LIN {X 0,Y 333.342,Z 944.319,A -85,B 0,C 180,E1 -9784.98,E2 -9784.98} C_VEL
LIN {X 0,Y 331.25,Z 957.354,A -85,B 0,C 180,E1 -9788.578,E2 -9788.578} C_VEL
LIN {X 0,Y 329.876,Z 968.022,A -85,B 0,C 180,E1 -9792.173,E2 -9792.173} C_VEL
LIN {X 0,Y 329.125,Z 976.186,A -85,B 0,C 180,E1 -9795.575,E2 -9795.575} C_VEL
LIN {X 0,Y 328.812,Z 982.598,A -85,B 0,C 180,E1 -9798.955,E2 -9798.955} C_VEL
LIN {X 0,Y 328.744,Z 987.468,A -85,B 0,C 180,E1 -9802.485,E2 -9802.485} C_VEL
LIN {X 0,Y 328.81,Z 990.364,A -85,B 0,C 180,E1 -9805.64,E2 -9805.64} C_VEL
LIN {X 0,Y 328.851,Z 991.822,A -85,B 0,C 180,E1 -9808.954,E2 -9808.954} C_VEL
LIN {X 0,Y 328.808,Z 991.751,A -85,B 0,C 180,E1 -9812.265,E2 -9812.265} C_VEL
LIN {X 0,Y 328.709,Z 990.204,A -85,B 0,C 180,E1 -9815.41,E2 -9815.41} C_VEL
LIN {X 0,Y 328.63,Z 986.844,A -85,B 0,C 180,E1 -9818.926,E2 -9818.926} C_VEL
LIN {X 0,Y 328.762,Z 981.971,A -85,B 0,C 180,E1 -9822.291,E2 -9822.291} C_VEL
LIN {X 0,Y 329.291,Z 975.055,A -85,B 0,C 180,E1 -9825.859,E2 -9825.859} C_VEL
LIN {X 0,Y 330.353,Z 966.159,A -85,B 0,C 180,E1 -9829.446,E2 -9829.446} C_VEL
LIN {X 0,Y 332.113,Z 955.071,A -85,B 0,C 180,E1 -9833.04,E2 -9833.04} C_VEL
LIN {X 0,Y 334.527,Z 942.274,A -85,B 0,C 180,E1 -9836.445,E2 -9836.445} C_VEL
LIN {X 0,Y 337.738,Z 926.952,A -85,B 0,C 180,E1 -9839.825,E2 -9839.825} C_VEL
LIN {X 0,Y 341.327,Z 910.684,A -85,B 0,C 180,E1 -9842.814,E2 -9842.814} C_VEL
LIN {X 0,Y 345.387,Z 892.681,A -85,B 0,C 180,E1 -9845.582,E2 -9845.582} C_VEL
LIN {X 0,Y 349.323,Z 874.881,A -85,B 0,C 180,E1 -9847.876,E2 -9847.876} C_VEL
LIN {X 0,Y 353.782,Z 854.185,A -85,B 0,C 180,E1 -9850.118,E2 -9850.118} C_VEL
LIN {X 0,Y 357.815,Z 834.405,A -85,B 0,C 180,E1 -9851.901,E2 -9851.901} C_VEL
LIN {X 0,Y 361.825,Z 812.887,A -85,B 0,C 180,E1 -9853.478,E2 -9853.478} C_VEL
LIN {X 0,Y 365.405,Z 791.398,A -85,B 0,C 180,E1 -9854.741,E2 -9854.741} C_VEL
LIN {X 0,Y 368.714,Z 768.497,A -85,B 0,C 180,E1 -9855.786,E2 -9855.786} C_VEL
LIN {X 0,Y 371.277,Z 745.338,A -85,B 0,C 180,E1 -9856.575,E2 -9856.575} C_VEL
LIN {X 0,Y 373.467,Z 717.783,A -85,B 0,C 180,E1 -9857.235,E2 -9857.235} C_VEL
LIN {X 0,Y 375.217,Z 704.776,A -85,B 0,C 180,E1 -9857.459,E2 -9857.459} C_VEL
LIN {X 0,Y 386.824,Z 676.005,A -85,B 0,C 180,E1 -9858.891,E2 -9858.891} C_VEL
LIN {X 0,Y 396.456,Z 655.426,A -85,B 0,C 180,E1 -9859.72,E2 -9859.72} C_VEL
LIN {X 0,Y 403.864,Z 640.656,A -85,B 0,C 180,E1 -9860.238,E2 -9860.238} C_VEL
LIN {X 0,Y 409.262,Z 629.343,A -85,B 0,C 180,E1 -9860.656,E2 -9860.656} C_VEL
LIN {X 0,Y 402.007,Z 613.046,A -85,B 0,C 180,E1 -9863.084,E2 -9863.084} C_VEL
LIN {X 0,Y 396.941,Z 595.631,A -85,B 0,C 180,E1 -9865.476,E2 -9865.476} C_VEL
LIN {X 0,Y 393.973,Z 576.533,A -85,B 0,C 180,E1 -9867.881,E2 -9867.881} C_VEL
LIN {X 0,Y 393.144,Z 556.331,A -85,B 0,C 180,E1 -9870.185,E2 -9870.185} C_VEL
LIN {X 0,Y 394.303,Z 535.428,A -85,B 0,C 180,E1 -9872.352,E2 -9872.352} C_VEL
LIN {X 0,Y 397.843,Z 510.824,A -85,B 0,C 180,E1 -9874.628,E2 -9874.628} C_VEL
LIN {X 0,Y 397.962,Z 509.912,A -85,B 0,C 180,E1 -9874.716,E2 -9874.716} C_VEL
LIN {X 0,Y 388.741,Z 492.166,A -85,B 0,C 180,E1 -9878.579,E2 -9878.579} C_VEL
LIN {X 0,Y 379.957,Z 475.806,A -85,B 0,C 180,E1 -9882.543,E2 -9882.543} C_VEL
LIN {X 0,Y 371.539,Z 460.665,A -85,B 0,C 180,E1 -9886.619,E2 -9886.619} C_VEL
LIN {X 0,Y 363.758,Z 446.974,A -85,B 0,C 180,E1 -9890.667,E2 -9890.667} C_VEL
LIN {X 0,Y 357.078,Z 435.672,A -85,B 0,C 180,E1 -9894.376,E2 -9894.376} C_VEL
LIN {X 0,Y 353.868,Z 430.258,A -85,B 0,C 180,E1 -9896.274,E2 -9896.274} C_VEL
LIN {X 0,Y 350.952,Z 425.333,A -85,B 0,C 180,E1 -9898.041,E2 -9898.041} C_VEL
LIN {X 0,Y 348.106,Z 420.507,A -85,B 0,C 180,E1 -9899.836,E2 -9899.836} C_VEL
LIN {X 0,Y 345.35,Z 415.775,A -85,B 0,C 180,E1 -9901.66,E2 -9901.66} C_VEL
LIN {X 0,Y 342.391,Z 410.76,A -85,B 0,C 180,E1 -9903.684,E2 -9903.684} C_VEL
LIN {X 0,Y 340.137,Z 407.168,A -85,B 0,C 180,E1 -9905.229,E2 -9905.229} C_VEL
LIN {X 0,Y 339.237,Z 405.463,A -85,B 0,C 180,E1 -9905.922,E2 -9905.922} C_VEL
LIN {X 0,Y 336.904,Z 401.699,A -85,B 0,C 180,E1 -9907.592,E2 -9907.592} C_VEL
LIN {X 0,Y 336.153,Z 400.24,A -85,B 0,C 180,E1 -9908.209,E2 -9908.209} C_VEL
LIN {X 0,Y 333.851,Z 396.936,A -85,B 0,C 180,E1 -9909.83,E2 -9909.83} C_VEL
LIN {X 0,Y 333.176,Z 395.055,A -85,B 0,C 180,E1 -9910.549,E2 -9910.549} C_VEL
LIN {X 0,Y 330.607,Z 391.768,A -85,B 0,C 180,E1 -9912.354,E2 -9912.354} C_VEL
LIN {X 0,Y 330.054,Z 389.618,A -85,B 0,C 180,E1 -9913.133,E2 -9913.133} C_VEL
LIN {X 0,Y 330.032,Z 389.621,A -85,B 0,C 180,E1 -9917.454,E2 -9917.454} C_VEL
LIN {X 0,Y 330.06,Z 389.619,A -85,B 0,C 180,E1 -9921.877,E2 -9921.877} C_VEL
LIN {X 0,Y 330.024,Z 389.616,A -85,B 0,C 180,E1 -9926.263,E2 -9926.263} C_VEL
LIN {X 0,Y 330.052,Z 389.609,A -85,B 0,C 180,E1 -9930.594,E2 -9930.594} C_VEL
LIN {X 0,Y 330.06,Z 389.802,A -85,B 0,C 180,E1 -9932.363,E2 -9932.363} C_VEL
LIN {X 0,Y 331.04,Z 392.665,A -85,B 0,C 180,E1 -9932.934,E2 -9932.934} C_VEL
LIN {X 0,Y 333.496,Z 395.723,A -85,B 0,C 180,E1 -9933.894,E2 -9933.894} C_VEL
LIN {X 0,Y 335.781,Z 399.63,A -85,B 0,C 180,E1 -9934.871,E2 -9934.871} C_VEL
LIN {X 0,Y 336.928,Z 401.545,A -85,B 0,C 180,E1 -9935.358,E2 -9935.358} C_VEL
LIN {X 0,Y 340.103,Z 406.895,A -85,B 0,C 180,E1 -9936.641,E2 -9936.641} C_VEL
LIN {X 0,Y 346.837,Z 418.945,A -85,B 0,C 180,E1 -9939.362,E2 -9939.362} C_VEL
LIN {X 0,Y 354.009,Z 433.623,A -85,B 0,C 180,E1 -9942.27,E2 -9942.27} C_VEL
LIN {X 0,Y 361.242,Z 450.647,A -85,B 0,C 180,E1 -9945.232,E2 -9945.232} C_VEL
LIN {X 0,Y 366.814,Z 465.9,A -85,B 0,C 180,E1 -9947.592,E2 -9947.592} C_VEL
LIN {X 0,Y 364.449,Z 505.857,A -85,B 0,C 180,E1 -9950.778,E2 -9950.778} C_VEL
LIN {X 0,Y 365.241,Z 514.351,A -85,B 0,C 180,E1 -9951.097,E2 -9951.097} C_VEL
LIN {X 0,Y 358.254,Z 708.662,A -85,B 0,C 180,E1 -9955.043,E2 -9955.043} C_VEL
LIN {X 0,Y 357.559,Z 727.861,A -85,B 0,C 180,E1 -9955.656,E2 -9955.656} C_VEL
LIN {X 0,Y 356.255,Z 746.186,A -85,B 0,C 180,E1 -9956.531,E2 -9956.531} C_VEL
LIN {X 0,Y 354.36,Z 763.972,A -85,B 0,C 180,E1 -9957.677,E2 -9957.677} C_VEL
LIN {X 0,Y 352.024,Z 780.749,A -85,B 0,C 180,E1 -9959.069,E2 -9959.069} C_VEL
LIN {X 0,Y 349.422,Z 796.485,A -85,B 0,C 180,E1 -9960.705,E2 -9960.705} C_VEL
LIN {X 0,Y 346.547,Z 811.319,A -85,B 0,C 180,E1 -9962.601,E2 -9962.601} C_VEL
LIN {X 0,Y 343.447,Z 825.625,A -85,B 0,C 180,E1 -9964.847,E2 -9964.847} C_VEL
LIN {X 0,Y 340.599,Z 837.864,A -85,B 0,C 180,E1 -9967.202,E2 -9967.202} C_VEL
LIN {X 0,Y 337.942,Z 848.709,A -85,B 0,C 180,E1 -9969.748,E2 -9969.748} C_VEL
LIN {X 0,Y 335.601,Z 858.18,A -85,B 0,C 180,E1 -9972.488,E2 -9972.488} C_VEL
LIN {X 0,Y 333.603,Z 866.416,A -85,B 0,C 180,E1 -9975.486,E2 -9975.486} C_VEL
LIN {X 0,Y 332.093,Z 872.879,A -85,B 0,C 180,E1 -9978.539,E2 -9978.539} C_VEL
LIN {X 0,Y 331.064,Z 877.731,A -85,B 0,C 180,E1 -9981.665,E2 -9981.665} C_VEL
LIN {X 0,Y 330.433,Z 881.111,A -85,B 0,C 180,E1 -9984.966,E2 -9984.966} C_VEL
LIN {X 0,Y 330.13,Z 882.813,A -85,B 0,C 180,E1 -9988.265,E2 -9988.265} C_VEL
LIN {X 0,Y 330.118,Z 882.889,A -85,B 0,C 180,E1 -9991.563,E2 -9991.563} C_VEL
LIN {X 0,Y 330.401,Z 881.34,A -85,B 0,C 180,E1 -9994.861,E2 -9994.861} C_VEL
LIN {X 0,Y 331.005,Z 878.106,A -85,B 0,C 180,E1 -9998.162,E2 -9998.162} C_VEL
LIN {X 0,Y 332.063,Z 873.069,A -85,B 0,C 180,E1 -10001.463,E2 -10001.463} C_VEL
LIN {X 0,Y 332.526,Z 871.056,A -85,B 0,C 180,E1 -10002.525,E2 -10002.525} C_VEL
LIN {X 0,Y 332.193,Z 868.673,A -85,B 0,C 180,E1 -10003.798,E2 -10003.798} C_VEL
LIN {X 0,Y 328.296,Z 862.096,A -85,B 0,C 180,E1 -10007.032,E2 -10007.032} C_VEL
LIN {X 0,Y 328.253,Z 858.758,A -85,B 0,C 180,E1 -10008.258,E2 -10008.258} C_VEL
LIN {X 0,Y 330.797,Z 849.028,A -85,B 0,C 180,E1 -10011.081,E2 -10011.081} C_VEL
LIN {X 0,Y 333.638,Z 837.979,A -85,B 0,C 180,E1 -10013.677,E2 -10013.677} C_VEL
LIN {X 0,Y 336.672,Z 825.502,A -85,B 0,C 180,E1 -10016.075,E2 -10016.075} C_VEL
LIN {X 0,Y 339.828,Z 811.487,A -85,B 0,C 180,E1 -10018.275,E2 -10018.275} C_VEL
LIN {X 0,Y 342.858,Z 796.414,A -85,B 0,C 180,E1 -10020.203,E2 -10020.203} C_VEL
LIN {X 0,Y 345.598,Z 780.325,A -85,B 0,C 180,E1 -10021.871,E2 -10021.871} C_VEL
LIN {X 0,Y 348.05,Z 763.099,A -85,B 0,C 180,E1 -10023.282,E2 -10023.282} C_VEL
LIN {X 0,Y 349.961,Z 744.96,A -85,B 0,C 180,E1 -10024.424,E2 -10024.424} C_VEL
LIN {X 0,Y 351.23,Z 726.587,A -85,B 0,C 180,E1 -10025.271,E2 -10025.271} C_VEL
LIN {X 0,Y 351.888,Z 707.076,A -85,B 0,C 180,E1 -10025.865,E2 -10025.865} C_VEL
LIN {X 0,Y 359.08,Z 513.009,A -85,B 0,C 180,E1 -10029.877,E2 -10029.877} C_VEL
LIN {X 0,Y 358.387,Z 506.854,A -85,B 0,C 180,E1 -10030.143,E2 -10030.143} C_VEL
LIN {X 0,Y 360.731,Z 469.551,A -85,B 0,C 180,E1 -10033.141,E2 -10033.141} C_VEL
LIN {X 0,Y 359.899,Z 467.043,A -85,B 0,C 180,E1 -10033.522,E2 -10033.522} C_VEL
LIN {X 0,Y 357.571,Z 466.596,A -85,B 0,C 180,E1 -10033.99,E2 -10033.99} C_VEL
LIN {X 0,Y 361.006,Z 476.688,A -85,B 0,C 180,E1 -10035.836,E2 -10035.836} C_VEL
LIN {X 0,Y 354.597,Z 519.378,A -85,B 0,C 180,E1 -10040.307,E2 -10040.307} C_VEL
LIN {X 0,Y 348.6,Z 563.579,A -85,B 0,C 180,E1 -10044.884,E2 -10044.884} C_VEL
LIN {X 0,Y 343.147,Z 608.894,A -85,B 0,C 180,E1 -10049.535,E2 -10049.535} C_VEL
LIN {X 0,Y 342.926,Z 612.486,A -85,B 0,C 180,E1 -10049.847,E2 -10049.847} C_VEL
LIN {X 0,Y 343.393,Z 622.189,A -85,B 0,C 180,E1 -10050.252,E2 -10050.252} C_VEL
LIN {X 0,Y 335.087,Z 752.809,A -85,B 0,C 180,E1 -10054.515,E2 -10054.515} C_VEL
LIN {X 0,Y 334.283,Z 770.76,A -85,B 0,C 180,E1 -10055.291,E2 -10055.291} C_VEL
LIN {X 0,Y 333.102,Z 788.151,A -85,B 0,C 180,E1 -10056.376,E2 -10056.376} C_VEL
LIN {X 0,Y 331.637,Z 804.493,A -85,B 0,C 180,E1 -10057.757,E2 -10057.757} C_VEL
LIN {X 0,Y 330.089,Z 819.19,A -85,B 0,C 180,E1 -10059.336,E2 -10059.336} C_VEL
LIN {X 0,Y 328.346,Z 834.099,A -85,B 0,C 180,E1 -10061.352,E2 -10061.352} C_VEL
LIN {X 0,Y 326.786,Z 846.627,A -85,B 0,C 180,E1 -10063.468,E2 -10063.468} C_VEL
LIN {X 0,Y 325.423,Z 857.745,A -85,B 0,C 180,E1 -10065.77,E2 -10065.77} C_VEL
LIN {X 0,Y 324.292,Z 867.369,A -85,B 0,C 180,E1 -10068.258,E2 -10068.258} C_VEL
LIN {X 0,Y 323.451,Z 875.603,A -85,B 0,C 180,E1 -10070.929,E2 -10070.929} C_VEL
LIN {X 0,Y 322.92,Z 882.228,A -85,B 0,C 180,E1 -10073.778,E2 -10073.778} C_VEL
LIN {X 0,Y 322.755,Z 887.037,A -85,B 0,C 180,E1 -10076.625,E2 -10076.625} C_VEL
LIN {X 0,Y 322.919,Z 890.358,A -85,B 0,C 180,E1 -10079.822,E2 -10079.822} C_VEL
LIN {X 0,Y 323.359,Z 891.535,A -85,B 0,C 180,E1 -10082.658,E2 -10082.658} C_VEL
LIN {X 0,Y 324.226,Z 891.056,A -85,B 0,C 180,E1 -10085.663,E2 -10085.663} C_VEL
LIN {X 0,Y 325.623,Z 888.514,A -85,B 0,C 180,E1 -10088.831,E2 -10088.831} C_VEL
LIN {X 0,Y 327.391,Z 884.461,A -85,B 0,C 180,E1 -10091.628,E2 -10091.628} C_VEL
LIN {X 0,Y 329.667,Z 878.673,A -85,B 0,C 180,E1 -10094.4,E2 -10094.4} C_VEL
LIN {X 0,Y 332.687,Z 870.277,A -85,B 0,C 180,E1 -10097.309,E2 -10097.309} C_VEL
LIN {X 0,Y 335.956,Z 860.542,A -85,B 0,C 180,E1 -10099.868,E2 -10099.868} C_VEL
LIN {X 0,Y 339.403,Z 849.527,A -85,B 0,C 180,E1 -10102.152,E2 -10102.152} C_VEL
LIN {X 0,Y 343.232,Z 836.315,A -85,B 0,C 180,E1 -10104.343,E2 -10104.343} C_VEL
LIN {X 0,Y 347.06,Z 821.915,A -85,B 0,C 180,E1 -10106.245,E2 -10106.245} C_VEL
LIN {X 0,Y 351.022,Z 805.964,A -85,B 0,C 180,E1 -10107.941,E2 -10107.941} C_VEL
LIN {X 0,Y 357.078,Z 783.037,A -85,B 0,C 180,E1 -10109.895,E2 -10109.895} C_VEL
LIN {X 0,Y 365.991,Z 756.399,A -85,B 0,C 180,E1 -10111.82,E2 -10111.82} C_VEL
LIN {X 0,Y 377.505,Z 723.16,A -85,B 0,C 180,E1 -10113.73,E2 -10113.73} C_VEL
LIN {X 0,Y 386.645,Z 693.172,A -85,B 0,C 180,E1 -10115.16,E2 -10115.16} C_VEL
LIN {X 0,Y 394.084,Z 667.225,A -85,B 0,C 180,E1 -10116.239,E2 -10116.239} C_VEL
LIN {X 0,Y 401.871,Z 655.163,A -85,B 0,C 180,E1 -10116.931,E2 -10116.931} C_VEL
LIN {X 0,Y 408.346,Z 646.955,A -85,B 0,C 180,E1 -10118.125,E2 -10118.125} C_VEL
LIN {X 0,Y 393.564,Z 674.807,A -85,B 0,C 180,E1 -10119.092,E2 -10119.092} C_VEL
LIN {X 0,Y 390.576,Z 686.577,A -85,B 0,C 180,E1 -10119.459,E2 -10119.459} C_VEL
LIN {X 0,Y 384.525,Z 712.431,A -85,B 0,C 180,E1 -10120.042,E2 -10120.042} C_VEL
LIN {X 0,Y 379.962,Z 730.467,A -85,B 0,C 180,E1 -10120.534,E2 -10120.534} C_VEL
LIN {X 0,Y 372.781,Z 758.728,A -85,B 0,C 180,E1 -10121.785,E2 -10121.785} C_VEL
LIN {X 0,Y 365.463,Z 785.63,A -85,B 0,C 180,E1 -10123.302,E2 -10123.302} C_VEL
LIN {X 0,Y 358.515,Z 810.818,A -85,B 0,C 180,E1 -10125.122,E2 -10125.122} C_VEL
LIN {X 0,Y 351.985,Z 834.7,A -85,B 0,C 180,E1 -10127.241,E2 -10127.241} C_VEL
LIN {X 0,Y 345.36,Z 859.368,A -85,B 0,C 180,E1 -10129.896,E2 -10129.896} C_VEL
LIN {X 0,Y 340.054,Z 879.999,A -85,B 0,C 180,E1 -10132.549,E2 -10132.549} C_VEL
LIN {X 0,Y 335.233,Z 899.403,A -85,B 0,C 180,E1 -10135.48,E2 -10135.48} C_VEL
LIN {X 0,Y 331.225,Z 916.555,A -85,B 0,C 180,E1 -10138.517,E2 -10138.517} C_VEL
LIN {X 0,Y 327.784,Z 932.46,A -85,B 0,C 180,E1 -10141.829,E2 -10141.829} C_VEL
LIN {X 0,Y 324.959,Z 947.091,A -85,B 0,C 180,E1 -10145.456,E2 -10145.456} C_VEL
LIN {X 0,Y 322.917,Z 959.714,A -85,B 0,C 180,E1 -10149.242,E2 -10149.242} C_VEL
LIN {X 0,Y 321.657,Z 969.925,A -85,B 0,C 180,E1 -10153.01,E2 -10153.01} C_VEL
LIN {X 0,Y 321.02,Z 977.806,A -85,B 0,C 180,E1 -10156.674,E2 -10156.674} C_VEL
LIN {X 0,Y 320.802,Z 983.523,A -85,B 0,C 180,E1 -10160.129,E2 -10160.129} C_VEL
LIN {X 0,Y 320.84,Z 987.541,A -85,B 0,C 180,E1 -10163.558,E2 -10163.558} C_VEL
LIN {X 0,Y 320.909,Z 989.98,A -85,B 0,C 180,E1 -10166.963,E2 -10166.963} C_VEL
LIN {X 0,Y 320.944,Z 990.779,A -85,B 0,C 180,E1 -10170.178,E2 -10170.178} C_VEL
LIN {X 0,Y 320.86,Z 990.107,A -85,B 0,C 180,E1 -10173.573,E2 -10173.573} C_VEL
LIN {X 0,Y 320.719,Z 987.806,A -85,B 0,C 180,E1 -10176.983,E2 -10176.983} C_VEL
LIN {X 0,Y 320.715,Z 983.933,A -85,B 0,C 180,E1 -10180.417,E2 -10180.417} C_VEL
LIN {X 0,Y 320.994,Z 978.022,A -85,B 0,C 180,E1 -10184.061,E2 -10184.061} C_VEL
LIN {X 0,Y 321.719,Z 970.64,A -85,B 0,C 180,E1 -10187.545,E2 -10187.545} C_VEL
LIN {X 0,Y 323.027,Z 961.408,A -85,B 0,C 180,E1 -10191.042,E2 -10191.042} C_VEL
LIN {X 0,Y 325.146,Z 949.445,A -85,B 0,C 180,E1 -10194.721,E2 -10194.721} C_VEL
LIN {X 0,Y 327.969,Z 935.671,A -85,B 0,C 180,E1 -10198.199,E2 -10198.199} C_VEL
LIN {X 0,Y 331.295,Z 920.762,A -85,B 0,C 180,E1 -10201.34,E2 -10201.34} C_VEL
LIN {X 0,Y 335.216,Z 903.919,A -85,B 0,C 180,E1 -10204.314,E2 -10204.314} C_VEL
LIN {X 0,Y 339.551,Z 885.243,A -85,B 0,C 180,E1 -10207.061,E2 -10207.061} C_VEL
LIN {X 0,Y 344.261,Z 864.347,A -85,B 0,C 180,E1 -10209.601,E2 -10209.601} C_VEL
LIN {X 0,Y 348.606,Z 844.573,A -85,B 0,C 180,E1 -10211.604,E2 -10211.604} C_VEL
LIN {X 0,Y 352.957,Z 823.133,A -85,B 0,C 180,E1 -10213.389,E2 -10213.389} C_VEL
LIN {X 0,Y 356.828,Z 801.846,A -85,B 0,C 180,E1 -10214.819,E2 -10214.819} C_VEL
LIN {X 0,Y 360.627,Z 778.349,A -85,B 0,C 180,E1 -10216.057,E2 -10216.057} C_VEL
LIN {X 0,Y 363.715,Z 755.272,A -85,B 0,C 180,E1 -10216.972,E2 -10216.972} C_VEL
LIN {X 0,Y 365.801,Z 731.561,A -85,B 0,C 180,E1 -10217.667,E2 -10217.667} C_VEL
LIN {X 0,Y 367.996,Z 710.151,A -85,B 0,C 180,E1 -10218.106,E2 -10218.106} C_VEL
LIN {X 0,Y 368.838,Z 704.318,A -85,B 0,C 180,E1 -10218.2,E2 -10218.2} C_VEL
LIN {X 0,Y 380.549,Z 675.592,A -85,B 0,C 180,E1 -10219.636,E2 -10219.636} C_VEL
LIN {X 0,Y 390.175,Z 655.218,A -85,B 0,C 180,E1 -10220.474,E2 -10220.474} C_VEL
LIN {X 0,Y 398.096,Z 639.628,A -85,B 0,C 180,E1 -10221.017,E2 -10221.017} C_VEL
LIN {X 0,Y 401.859,Z 631.602,A -85,B 0,C 180,E1 -10221.325,E2 -10221.325} C_VEL
LIN {X 0,Y 394.83,Z 614.668,A -85,B 0,C 180,E1 -10223.84,E2 -10223.84} C_VEL
LIN {X 0,Y 390.221,Z 597.312,A -85,B 0,C 180,E1 -10226.22,E2 -10226.22} C_VEL
LIN {X 0,Y 387.565,Z 578.081,A -85,B 0,C 180,E1 -10228.641,E2 -10228.641} C_VEL
LIN {X 0,Y 387.071,Z 557.241,A -85,B 0,C 180,E1 -10231.031,E2 -10231.031} C_VEL
LIN {X 0,Y 388.574,Z 535.98,A -85,B 0,C 180,E1 -10233.237,E2 -10233.237} C_VEL
LIN {X 0,Y 391.857,Z 514.196,A -85,B 0,C 180,E1 -10235.263,E2 -10235.263} C_VEL
LIN {X 0,Y 383.368,Z 497.684,A -85,B 0,C 180,E1 -10238.905,E2 -10238.905} C_VEL
LIN {X 0,Y 374.539,Z 481.229,A -85,B 0,C 180,E1 -10242.924,E2 -10242.924} C_VEL
LIN {X 0,Y 366.427,Z 466.54,A -85,B 0,C 180,E1 -10246.911,E2 -10246.911} C_VEL
LIN {X 0,Y 358.659,Z 452.809,A -85,B 0,C 180,E1 -10251.019,E2 -10251.019} C_VEL
LIN {X 0,Y 351.921,Z 441.384,A -85,B 0,C 180,E1 -10254.784,E2 -10254.784} C_VEL
LIN {X 0,Y 348.681,Z 435.902,A -85,B 0,C 180,E1 -10256.713,E2 -10256.713} C_VEL
LIN {X 0,Y 345.807,Z 430.994,A -85,B 0,C 180,E1 -10258.509,E2 -10258.509} C_VEL
LIN {X 0,Y 343.227,Z 426.58,A -85,B 0,C 180,E1 -10260.167,E2 -10260.167} C_VEL
LIN {X 0,Y 340.412,Z 421.817,A -85,B 0,C 180,E1 -10262.02,E2 -10262.02} C_VEL
LIN {X 0,Y 337.395,Z 416.778,A -85,B 0,C 180,E1 -10264.079,E2 -10264.079} C_VEL
LIN {X 0,Y 335.066,Z 412.505,A -85,B 0,C 180,E1 -10265.824,E2 -10265.824} C_VEL
LIN {X 0,Y 332.326,Z 408.24,A -85,B 0,C 180,E1 -10267.782,E2 -10267.782} C_VEL
LIN {X 0,Y 331.376,Z 406.559,A -85,B 0,C 180,E1 -10268.503,E2 -10268.503} C_VEL
LIN {X 0,Y 328.991,Z 402.694,A -85,B 0,C 180,E1 -10270.33,E2 -10270.33} C_VEL
LIN {X 0,Y 328.052,Z 401.087,A -85,B 0,C 180,E1 -10271.067,E2 -10271.067} C_VEL
LIN {X 0,Y 325.86,Z 397.789,A -85,B 0,C 180,E1 -10272.764,E2 -10272.764} C_VEL
LIN {X 0,Y 325.032,Z 395.848,A -85,B 0,C 180,E1 -10273.574,E2 -10273.574} C_VEL
LIN {X 0,Y 322.788,Z 392.975,A -85,B 0,C 180,E1 -10275.266,E2 -10275.266} C_VEL
LIN {X 0,Y 322.094,Z 390.61,A -85,B 0,C 180,E1 -10276.224,E2 -10276.224} C_VEL
LIN {X 0,Y 322.11,Z 390.604,A -85,B 0,C 180,E1 -10280.915,E2 -10280.915} C_VEL
LIN {X 0,Y 322.083,Z 390.617,A -85,B 0,C 180,E1 -10285.397,E2 -10285.397} C_VEL
LIN {X 0,Y 322.114,Z 390.612,A -85,B 0,C 180,E1 -10289.643,E2 -10289.643} C_VEL
LIN {X 0,Y 322.126,Z 390.626,A -85,B 0,C 180,E1 -10290.312,E2 -10290.312} C_VEL
LIN {X 0,Y 323.043,Z 393.495,A -85,B 0,C 180,E1 -10290.917,E2 -10290.917} C_VEL
LIN {X 0,Y 325.472,Z 396.18,A -85,B 0,C 180,E1 -10291.897,E2 -10291.897} C_VEL
LIN {X 0,Y 327.525,Z 400.234,A -85,B 0,C 180,E1 -10292.916,E2 -10292.916} C_VEL
LIN {X 0,Y 329.128,Z 402.367,A -85,B 0,C 180,E1 -10293.567,E2 -10293.567} C_VEL
LIN {X 0,Y 332.527,Z 408.079,A -85,B 0,C 180,E1 -10295.052,E2 -10295.052} C_VEL
LIN {X 0,Y 337.194,Z 416.006,A -85,B 0,C 180,E1 -10297.01,E2 -10297.01} C_VEL
LIN {X 0,Y 344.143,Z 429.404,A -85,B 0,C 180,E1 -10299.948,E2 -10299.948} C_VEL
LIN {X 0,Y 350.801,Z 443.734,A -85,B 0,C 180,E1 -10302.716,E2 -10302.716} C_VEL
LIN {X 0,Y 357.748,Z 461.185,A -85,B 0,C 180,E1 -10305.684,E2 -10305.684} C_VEL
LIN {X 0,Y 360.649,Z 469.904,A -85,B 0,C 180,E1 -10307,E2 -10307} C_VEL
LIN {X 0,Y 358.347,Z 507.3,A -85,B 0,C 180,E1 -10309.985,E2 -10309.985} C_VEL
LIN {X 0,Y 359.086,Z 515.499,A -85,B 0,C 180,E1 -10310.3,E2 -10310.3} C_VEL
LIN {X 0,Y 351.79,Z 709.225,A -85,B 0,C 180,E1 -10314.288,E2 -10314.288} C_VEL
LIN {X 0,Y 351.081,Z 728.581,A -85,B 0,C 180,E1 -10314.906,E2 -10314.906} C_VEL
LIN {X 0,Y 349.757,Z 746.717,A -85,B 0,C 180,E1 -10315.775,E2 -10315.775} C_VEL
LIN {X 0,Y 347.856,Z 764.136,A -85,B 0,C 180,E1 -10316.899,E2 -10316.899} C_VEL
LIN {X 0,Y 345.564,Z 780.231,A -85,B 0,C 180,E1 -10318.224,E2 -10318.224} C_VEL
LIN {X 0,Y 342.826,Z 796.335,A -85,B 0,C 180,E1 -10319.892,E2 -10319.892} C_VEL
LIN {X 0,Y 339.769,Z 811.562,A -85,B 0,C 180,E1 -10321.84,E2 -10321.84} C_VEL
LIN {X 0,Y 336.765,Z 824.956,A -85,B 0,C 180,E1 -10323.934,E2 -10323.934} C_VEL
LIN {X 0,Y 333.72,Z 837.525,A -85,B 0,C 180,E1 -10326.33,E2 -10326.33} C_VEL
LIN {X 0,Y 330.869,Z 848.651,A -85,B 0,C 180,E1 -10328.924,E2 -10328.924} C_VEL
LIN {X 0,Y 328.332,Z 858.368,A -85,B 0,C 180,E1 -10331.72,E2 -10331.72} C_VEL
LIN {X 0,Y 326.085,Z 867.09,A -85,B 0,C 180,E1 -10334.893,E2 -10334.893} C_VEL
LIN {X 0,Y 324.408,Z 873.817,A -85,B 0,C 180,E1 -10338.083,E2 -10338.083} C_VEL
LIN {X 0,Y 323.28,Z 878.762,A -85,B 0,C 180,E1 -10341.284,E2 -10341.284} C_VEL
LIN {X 0,Y 322.582,Z 882.228,A -85,B 0,C 180,E1 -10344.665,E2 -10344.665} C_VEL
LIN {X 0,Y 322.242,Z 884.013,A -85,B 0,C 180,E1 -10348.045,E2 -10348.045} C_VEL
LIN {X 0,Y 322.209,Z 884.173,A -85,B 0,C 180,E1 -10351.423,E2 -10351.423} C_VEL
LIN {X 0,Y 322.497,Z 882.711,A -85,B 0,C 180,E1 -10354.802,E2 -10354.802} C_VEL
LIN {X 0,Y 323.126,Z 879.588,A -85,B 0,C 180,E1 -10358.184,E2 -10358.184} C_VEL
LIN {X 0,Y 324.232,Z 874.663,A -85,B 0,C 180,E1 -10361.564,E2 -10361.564} C_VEL
LIN {X 0,Y 325.829,Z 868.196,A -85,B 0,C 180,E1 -10364.756,E2 -10364.756} C_VEL
LIN {X 0,Y 327.861,Z 860.296,A -85,B 0,C 180,E1 -10367.757,E2 -10367.757} C_VEL
LIN {X 0,Y 328.253,Z 858.758,A -85,B 0,C 180,E1 -10368.258,E2 -10368.258} C_VEL
LIN {X 0,Y 328.312,Z 855.247,A -85,B 0,C 180,E1 -10369.468,E2 -10369.468} C_VEL
LIN {X 0,Y 325.569,Z 846.681,A -85,B 0,C 180,E1 -10372.406,E2 -10372.406} C_VEL
LIN {X 0,Y 325.608,Z 842.379,A -85,B 0,C 180,E1 -10373.543,E2 -10373.543} C_VEL
LIN {X 0,Y 325.759,Z 841.698,A -85,B 0,C 180,E1 -10373.695,E2 -10373.695} C_VEL
LIN {X 0,Y 328.87,Z 829.649,A -85,B 0,C 180,E1 -10376.158,E2 -10376.158} C_VEL
LIN {X 0,Y 332.096,Z 816.217,A -85,B 0,C 180,E1 -10378.405,E2 -10378.405} C_VEL
LIN {X 0,Y 335.202,Z 801.871,A -85,B 0,C 180,E1 -10380.371,E2 -10380.371} C_VEL
LIN {X 0,Y 338.18,Z 785.864,A -85,B 0,C 180,E1 -10382.154,E2 -10382.154} C_VEL
LIN {X 0,Y 340.843,Z 768.715,A -85,B 0,C 180,E1 -10383.672,E2 -10383.672} C_VEL
LIN {X 0,Y 342.994,Z 750.871,A -85,B 0,C 180,E1 -10384.896,E2 -10384.896} C_VEL
LIN {X 0,Y 344.507,Z 732.515,A -85,B 0,C 180,E1 -10385.835,E2 -10385.835} C_VEL
LIN {X 0,Y 345.338,Z 713.77,A -85,B 0,C 180,E1 -10386.493,E2 -10386.493} C_VEL
LIN {X 0,Y 347.277,Z 656.18,A -85,B 0,C 180,E1 -10387.751,E2 -10387.751} C_VEL
LIN {X 0,Y 353,Z 514.152,A -85,B 0,C 180,E1 -10390.705,E2 -10390.705} C_VEL
LIN {X 0,Y 352.344,Z 507.898,A -85,B 0,C 180,E1 -10390.988,E2 -10390.988} C_VEL
LIN {X 0,Y 354.472,Z 474.28,A -85,B 0,C 180,E1 -10393.713,E2 -10393.713} C_VEL
LIN {X 0,Y 352.418,Z 473.833,A -85,B 0,C 180,E1 -10394.126,E2 -10394.126} C_VEL
LIN {X 0,Y 354.449,Z 480.013,A -85,B 0,C 180,E1 -10395.266,E2 -10395.266} C_VEL
LIN {X 0,Y 347.909,Z 522.053,A -85,B 0,C 180,E1 -10399.711,E2 -10399.711} C_VEL
LIN {X 0,Y 341.735,Z 565.667,A -85,B 0,C 180,E1 -10404.288,E2 -10404.288} C_VEL
LIN {X 0,Y 336.039,Z 611.159,A -85,B 0,C 180,E1 -10409.019,E2 -10409.019} C_VEL
LIN {X 0,Y 336.01,Z 613.936,A -85,B 0,C 180,E1 -10409.214,E2 -10409.214} C_VEL
LIN {X 0,Y 336.383,Z 623.109,A -85,B 0,C 180,E1 -10409.611,E2 -10409.611} C_VEL
LIN {X 0,Y 327.812,Z 750.237,A -85,B 0,C 180,E1 -10413.885,E2 -10413.885} C_VEL
LIN {X 0,Y 326.89,Z 770.292,A -85,B 0,C 180,E1 -10414.742,E2 -10414.742} C_VEL
LIN {X 0,Y 325.605,Z 788.541,A -85,B 0,C 180,E1 -10415.894,E2 -10415.894} C_VEL
LIN {X 0,Y 324.115,Z 804.77,A -85,B 0,C 180,E1 -10417.278,E2 -10417.278} C_VEL
LIN {X 0,Y 322.424,Z 820.328,A -85,B 0,C 180,E1 -10418.976,E2 -10418.976} C_VEL
LIN {X 0,Y 320.591,Z 835.475,A -85,B 0,C 180,E1 -10421.073,E2 -10421.073} C_VEL
LIN {X 0,Y 318.982,Z 847.994,A -85,B 0,C 180,E1 -10423.239,E2 -10423.239} C_VEL
LIN {X 0,Y 317.571,Z 859.083,A -85,B 0,C 180,E1 -10425.597,E2 -10425.597} C_VEL
LIN {X 0,Y 316.402,Z 868.699,A -85,B 0,C 180,E1 -10428.146,E2 -10428.146} C_VEL
LIN {X 0,Y 315.542,Z 876.956,A -85,B 0,C 180,E1 -10430.883,E2 -10430.883} C_VEL
LIN {X 0,Y 315.007,Z 883.627,A -85,B 0,C 180,E1 -10433.804,E2 -10433.804} C_VEL
LIN {X 0,Y 314.854,Z 888.469,A -85,B 0,C 180,E1 -10436.723,E2 -10436.723} C_VEL
LIN {X 0,Y 315.058,Z 891.838,A -85,B 0,C 180,E1 -10439.999,E2 -10439.999} C_VEL
LIN {X 0,Y 315.597,Z 893.086,A -85,B 0,C 180,E1 -10443.087,E2 -10443.087} C_VEL
LIN {X 0,Y 316.573,Z 892.557,A -85,B 0,C 180,E1 -10446.164,E2 -10446.164} C_VEL
LIN {X 0,Y 318.152,Z 890.012,A -85,B 0,C 180,E1 -10449.405,E2 -10449.405} C_VEL
LIN {X 0,Y 320.384,Z 885.342,A -85,B 0,C 180,E1 -10452.618,E2 -10452.618} C_VEL
LIN {X 0,Y 323.12,Z 878.836,A -85,B 0,C 180,E1 -10455.617,E2 -10455.617} C_VEL
LIN {X 0,Y 326.097,Z 871.213,A -85,B 0,C 180,E1 -10458.224,E2 -10458.224} C_VEL
LIN {X 0,Y 329.393,Z 862.35,A -85,B 0,C 180,E1 -10460.616,E2 -10460.616} C_VEL
LIN {X 0,Y 333.177,Z 851.404,A -85,B 0,C 180,E1 -10462.962,E2 -10462.962} C_VEL
LIN {X 0,Y 337.471,Z 837.953,A -85,B 0,C 180,E1 -10465.254,E2 -10465.254} C_VEL
LIN {X 0,Y 341.655,Z 823.96,A -85,B 0,C 180,E1 -10467.168,E2 -10467.168} C_VEL
LIN {X 0,Y 346.212,Z 808.13,A -85,B 0,C 180,E1 -10468.929,E2 -10468.929} C_VEL
LIN {X 0,Y 352.822,Z 786.676,A -85,B 0,C 180,E1 -10470.859,E2 -10470.859} C_VEL
LIN {X 0,Y 362.226,Z 761.67,A -85,B 0,C 180,E1 -10472.753,E2 -10472.753} C_VEL
LIN {X 0,Y 372.998,Z 733.507,A -85,B 0,C 180,E1 -10474.444,E2 -10474.444} C_VEL
LIN {X 0,Y 382.553,Z 705.665,A -85,B 0,C 180,E1 -10475.835,E2 -10475.835} C_VEL
LIN {X 0,Y 393.309,Z 670.237,A -85,B 0,C 180,E1 -10477.323,E2 -10477.323} C_VEL
LIN {X 0,Y 396.762,Z 665.045,A -85,B 0,C 180,E1 -10477.589,E2 -10477.589} C_VEL
LIN {X 0,Y 392.506,Z 673.483,A -85,B 0,C 180,E1 -10477.888,E2 -10477.888} C_VEL
LIN {X 0,Y 386.708,Z 696.319,A -85,B 0,C 180,E1 -10478.543,E2 -10478.543} C_VEL
LIN {X 0,Y 378.769,Z 725.834,A -85,B 0,C 180,E1 -10479.215,E2 -10479.215} C_VEL
LIN {X 0,Y 372.596,Z 747.779,A -85,B 0,C 180,E1 -10480.11,E2 -10480.11} C_VEL
LIN {X 0,Y 364.607,Z 774.728,A -85,B 0,C 180,E1 -10481.526,E2 -10481.526} C_VEL
LIN {X 0,Y 357.097,Z 799.271,A -85,B 0,C 180,E1 -10483.164,E2 -10483.164} C_VEL
LIN {X 0,Y 349.742,Z 823.445,A -85,B 0,C 180,E1 -10485.182,E2 -10485.182} C_VEL
LIN {X 0,Y 342.197,Z 848.824,A -85,B 0,C 180,E1 -10487.775,E2 -10487.775} C_VEL
LIN {X 0,Y 335.792,Z 871.104,A -85,B 0,C 180,E1 -10490.526,E2 -10490.526} C_VEL
LIN {X 0,Y 330.069,Z 891.923,A -85,B 0,C 180,E1 -10493.577,E2 -10493.577} C_VEL
LIN {X 0,Y 325.223,Z 910.63,A -85,B 0,C 180,E1 -10496.822,E2 -10496.822} C_VEL
LIN {X 0,Y 321.341,Z 926.875,A -85,B 0,C 180,E1 -10500.142,E2 -10500.142} C_VEL
LIN {X 0,Y 318.282,Z 941.016,A -85,B 0,C 180,E1 -10503.547,E2 -10503.547} C_VEL
LIN {X 0,Y 315.839,Z 954.038,A -85,B 0,C 180,E1 -10507.28,E2 -10507.28} C_VEL
LIN {X 0,Y 314.149,Z 965.376,A -85,B 0,C 180,E1 -10511.248,E2 -10511.248} C_VEL
LIN {X 0,Y 313.244,Z 973.977,A -85,B 0,C 180,E1 -10515.016,E2 -10515.016} C_VEL
LIN {X 0,Y 312.908,Z 980.358,A -85,B 0,C 180,E1 -10518.573,E2 -10518.573} C_VEL
LIN {X 0,Y 312.869,Z 985.233,A -85,B 0,C 180,E1 -10522.286,E2 -10522.286} C_VEL
LIN {X 0,Y 312.967,Z 988.052,A -85,B 0,C 180,E1 -10525.602,E2 -10525.602} C_VEL
LIN {X 0,Y 313.028,Z 989.46,A -85,B 0,C 180,E1 -10529.084,E2 -10529.084} C_VEL
LIN {X 0,Y 312.98,Z 989.327,A -85,B 0,C 180,E1 -10532.38,E2 -10532.38} C_VEL
LIN {X 0,Y 312.866,Z 987.705,A -85,B 0,C 180,E1 -10535.685,E2 -10535.685} C_VEL
LIN {X 0,Y 312.753,Z 984.452,A -85,B 0,C 180,E1 -10539.198,E2 -10539.198} C_VEL
LIN {X 0,Y 312.894,Z 979.501,A -85,B 0,C 180,E1 -10542.737,E2 -10542.737} C_VEL
LIN {X 0,Y 313.435,Z 972.859,A -85,B 0,C 180,E1 -10546.303,E2 -10546.303} C_VEL
LIN {X 0,Y 314.595,Z 963.883,A -85,B 0,C 180,E1 -10550.074,E2 -10550.074} C_VEL
LIN {X 0,Y 316.524,Z 952.684,A -85,B 0,C 180,E1 -10553.849,E2 -10553.849} C_VEL
LIN {X 0,Y 319.174,Z 939.755,A -85,B 0,C 180,E1 -10557.419,E2 -10557.419} C_VEL
LIN {X 0,Y 322.571,Z 924.748,A -85,B 0,C 180,E1 -10560.841,E2 -10560.841} C_VEL
LIN {X 0,Y 326.496,Z 908.231,A -85,B 0,C 180,E1 -10563.978,E2 -10563.978} C_VEL
LIN {X 0,Y 330.733,Z 890.69,A -85,B 0,C 180,E1 -10566.768,E2 -10566.768} C_VEL
LIN {X 0,Y 334.977,Z 872.792,A -85,B 0,C 180,E1 -10569.145,E2 -10569.145} C_VEL
LIN {X 0,Y 339.759,Z 851.968,A -85,B 0,C 180,E1 -10571.463,E2 -10571.463} C_VEL
LIN {X 0,Y 344.234,Z 831.32,A -85,B 0,C 180,E1 -10573.364,E2 -10573.364} C_VEL
LIN {X 0,Y 348.583,Z 809.506,A -85,B 0,C 180,E1 -10574.995,E2 -10574.995} C_VEL
LIN {X 0,Y 352.516,Z 787.036,A -85,B 0,C 180,E1 -10576.325,E2 -10576.325} C_VEL
LIN {X 0,Y 356.033,Z 763.708,A -85,B 0,C 180,E1 -10577.379,E2 -10577.379} C_VEL
LIN {X 0,Y 358.665,Z 739.823,A -85,B 0,C 180,E1 -10578.183,E2 -10578.183} C_VEL
LIN {X 0,Y 360.776,Z 716.305,A -85,B 0,C 180,E1 -10578.749,E2 -10578.749} C_VEL
LIN {X 0,Y 362.628,Z 703.337,A -85,B 0,C 180,E1 -10578.977,E2 -10578.977} C_VEL
LIN {X 0,Y 374.76,Z 674.162,A -85,B 0,C 180,E1 -10580.448,E2 -10580.448} C_VEL
LIN {X 0,Y 384.936,Z 652.913,A -85,B 0,C 180,E1 -10581.309,E2 -10581.309} C_VEL
LIN {X 0,Y 392.877,Z 637.446,A -85,B 0,C 180,E1 -10581.849,E2 -10581.849} C_VEL
LIN {X 0,Y 394.546,Z 633.89,A -85,B 0,C 180,E1 -10581.99,E2 -10581.99} C_VEL
LIN {X 0,Y 387.855,Z 616.662,A -85,B 0,C 180,E1 -10584.549,E2 -10584.549} C_VEL
LIN {X 0,Y 383.54,Z 598.909,A -85,B 0,C 180,E1 -10586.986,E2 -10586.986} C_VEL
LIN {X 0,Y 381.256,Z 579.69,A -85,B 0,C 180,E1 -10589.418,E2 -10589.418} C_VEL
LIN {X 0,Y 381.038,Z 558.125,A -85,B 0,C 180,E1 -10591.892,E2 -10591.892} C_VEL
LIN {X 0,Y 382.885,Z 536.402,A -85,B 0,C 180,E1 -10594.145,E2 -10594.145} C_VEL
LIN {X 0,Y 385.742,Z 518.393,A -85,B 0,C 180,E1 -10595.838,E2 -10595.838} C_VEL
LIN {X 0,Y 376.651,Z 500.701,A -85,B 0,C 180,E1 -10599.813,E2 -10599.813} C_VEL
LIN {X 0,Y 368.508,Z 485.577,A -85,B 0,C 180,E1 -10603.61,E2 -10603.61} C_VEL
LIN {X 0,Y 361.287,Z 472.385,A -85,B 0,C 180,E1 -10607.209,E2 -10607.209} C_VEL
LIN {X 0,Y 353.472,Z 458.565,A -85,B 0,C 180,E1 -10611.378,E2 -10611.378} C_VEL
LIN {X 0,Y 347.063,Z 447.542,A -85,B 0,C 180,E1 -10615.042,E2 -10615.042} C_VEL
LIN {X 0,Y 342.018,Z 438.737,A -85,B 0,C 180,E1 -10618.158,E2 -10618.158} C_VEL
LIN {X 0,Y 336.152,Z 428.72,A -85,B 0,C 180,E1 -10621.986,E2 -10621.986} C_VEL
LIN {X 0,Y 332.431,Z 422.772,A -85,B 0,C 180,E1 -10624.486,E2 -10624.486} C_VEL
LIN {X 0,Y 329.762,Z 418.099,A -85,B 0,C 180,E1 -10626.442,E2 -10626.442} C_VEL
LIN {X 0,Y 327.358,Z 413.918,A -85,B 0,C 180,E1 -10628.272,E2 -10628.272} C_VEL
LIN {X 0,Y 324.392,Z 409.239,A -85,B 0,C 180,E1 -10630.507,E2 -10630.507} C_VEL
LIN {X 0,Y 323.544,Z 407.639,A -85,B 0,C 180,E1 -10631.227,E2 -10631.227} C_VEL
LIN {X 0,Y 321.123,Z 403.881,A -85,B 0,C 180,E1 -10633.138,E2 -10633.138} C_VEL
LIN {X 0,Y 320.286,Z 402.205,A -85,B 0,C 180,E1 -10633.909,E2 -10633.909} C_VEL
LIN {X 0,Y 318.043,Z 399.002,A -85,B 0,C 180,E1 -10635.687,E2 -10635.687} C_VEL
LIN {X 0,Y 317.193,Z 396.948,A -85,B 0,C 180,E1 -10636.612,E2 -10636.612} C_VEL
LIN {X 0,Y 314.786,Z 393.908,A -85,B 0,C 180,E1 -10638.52,E2 -10638.52} C_VEL
LIN {X 0,Y 314.168,Z 391.603,A -85,B 0,C 180,E1 -10639.523,E2 -10639.523} C_VEL
LIN {X 0,Y 314.17,Z 391.592,A -85,B 0,C 180,E1 -10643.84,E2 -10643.84} C_VEL
LIN {X 0,Y 314.177,Z 391.599,A -85,B 0,C 180,E1 -10648.034,E2 -10648.034} C_VEL
LIN {X 0,Y 315.333,Z 394.855,A -85,B 0,C 180,E1 -10648.814,E2 -10648.814} C_VEL
LIN {X 0,Y 317.99,Z 397.874,A -85,B 0,C 180,E1 -10649.997,E2 -10649.997} C_VEL
LIN {X 0,Y 319.961,Z 401.551,A -85,B 0,C 180,E1 -10651.039,E2 -10651.039} C_VEL
LIN {X 0,Y 321.183,Z 402.791,A -85,B 0,C 180,E1 -10651.534,E2 -10651.534} C_VEL
LIN {X 0,Y 323.248,Z 406.693,A -85,B 0,C 180,E1 -10652.563,E2 -10652.563} C_VEL
LIN {X 0,Y 324.801,Z 408.913,A -85,B 0,C 180,E1 -10653.227,E2 -10653.227} C_VEL
LIN {X 0,Y 330.074,Z 417.703,A -85,B 0,C 180,E1 -10655.564,E2 -10655.564} C_VEL
LIN {X 0,Y 337.28,Z 431.359,A -85,B 0,C 180,E1 -10658.72,E2 -10658.72} C_VEL
LIN {X 0,Y 344.17,Z 446.06,A -85,B 0,C 180,E1 -10661.704,E2 -10661.704} C_VEL
LIN {X 0,Y 350.852,Z 462.505,A -85,B 0,C 180,E1 -10664.627,E2 -10664.627} C_VEL
LIN {X 0,Y 354.576,Z 473.016,A -85,B 0,C 180,E1 -10666.302,E2 -10666.302} C_VEL
LIN {X 0,Y 352.312,Z 508.73,A -85,B 0,C 180,E1 -10669.164,E2 -10669.164} C_VEL
LIN {X 0,Y 352.999,Z 516.773,A -85,B 0,C 180,E1 -10669.478,E2 -10669.478} C_VEL
LIN {X 0,Y 345.39,Z 709.668,A -85,B 0,C 180,E1 -10673.502,E2 -10673.502} C_VEL
LIN {X 0,Y 344.662,Z 729.248,A -85,B 0,C 180,E1 -10674.127,E2 -10674.127} C_VEL
LIN {X 0,Y 343.246,Z 747.952,A -85,B 0,C 180,E1 -10675.032,E2 -10675.032} C_VEL
LIN {X 0,Y 341.262,Z 765.38,A -85,B 0,C 180,E1 -10676.174,E2 -10676.174} C_VEL
LIN {X 0,Y 338.771,Z 782.06,A -85,B 0,C 180,E1 -10677.577,E2 -10677.577} C_VEL
LIN {X 0,Y 336.013,Z 797.589,A -85,B 0,C 180,E1 -10679.216,E2 -10679.216} C_VEL
LIN {X 0,Y 332.917,Z 812.4,A -85,B 0,C 180,E1 -10681.136,E2 -10681.136} C_VEL
LIN {X 0,Y 329.677,Z 826.217,A -85,B 0,C 180,E1 -10683.33,E2 -10683.33} C_VEL
LIN {X 0,Y 326.485,Z 838.788,A -85,B 0,C 180,E1 -10685.772,E2 -10685.772} C_VEL
LIN {X 0,Y 323.49,Z 849.916,A -85,B 0,C 180,E1 -10688.42,E2 -10688.42} C_VEL
LIN {X 0,Y 320.716,Z 859.998,A -85,B 0,C 180,E1 -10691.397,E2 -10691.397} C_VEL
LIN {X 0,Y 318.393,Z 868.54,A -85,B 0,C 180,E1 -10694.599,E2 -10694.599} C_VEL
LIN {X 0,Y 316.661,Z 875.084,A -85,B 0,C 180,E1 -10697.787,E2 -10697.787} C_VEL
LIN {X 0,Y 315.457,Z 880.029,A -85,B 0,C 180,E1 -10701.066,E2 -10701.066} C_VEL
LIN {X 0,Y 314.709,Z 883.493,A -85,B 0,C 180,E1 -10704.531,E2 -10704.531} C_VEL
LIN {X 0,Y 314.346,Z 885.277,A -85,B 0,C 180,E1 -10707.995,E2 -10707.995} C_VEL
LIN {X 0,Y 314.312,Z 885.436,A -85,B 0,C 180,E1 -10711.459,E2 -10711.459} C_VEL
LIN {X 0,Y 314.619,Z 883.975,A -85,B 0,C 180,E1 -10714.923,E2 -10714.923} C_VEL
LIN {X 0,Y 315.293,Z 880.852,A -85,B 0,C 180,E1 -10718.389,E2 -10718.389} C_VEL
LIN {X 0,Y 316.473,Z 875.928,A -85,B 0,C 180,E1 -10721.851,E2 -10721.851} C_VEL
LIN {X 0,Y 318.171,Z 869.46,A -85,B 0,C 180,E1 -10725.12,E2 -10725.12} C_VEL
LIN {X 0,Y 320.321,Z 861.559,A -85,B 0,C 180,E1 -10728.189,E2 -10728.189} C_VEL
LIN {X 0,Y 322.88,Z 852.275,A -85,B 0,C 180,E1 -10731.053,E2 -10731.053} C_VEL
LIN {X 0,Y 325.759,Z 841.698,A -85,B 0,C 180,E1 -10733.695,E2 -10733.695} C_VEL
LIN {X 0,Y 326.081,Z 837.195,A -85,B 0,C 180,E1 -10734.789,E2 -10734.789} C_VEL
LIN {X 0,Y 324.002,Z 825.51,A -85,B 0,C 180,E1 -10737.656,E2 -10737.656} C_VEL
LIN {X 0,Y 324.528,Z 820.124,A -85,B 0,C 180,E1 -10738.655,E2 -10738.655} C_VEL
LIN {X 0,Y 327.982,Z 805.209,A -85,B 0,C 180,E1 -10740.808,E2 -10740.808} C_VEL
LIN {X 0,Y 331.07,Z 789.683,A -85,B 0,C 180,E1 -10742.622,E2 -10742.622} C_VEL
LIN {X 0,Y 333.835,Z 773.181,A -85,B 0,C 180,E1 -10744.165,E2 -10744.165} C_VEL
LIN {X 0,Y 336.161,Z 755.605,A -85,B 0,C 180,E1 -10745.451,E2 -10745.451} C_VEL
LIN {X 0,Y 337.857,Z 737.511,A -85,B 0,C 180,E1 -10746.449,E2 -10746.449} C_VEL
LIN {X 0,Y 338.864,Z 718.985,A -85,B 0,C 180,E1 -10747.169,E2 -10747.169} C_VEL
LIN {X 0,Y 340.107,Z 679.343,A -85,B 0,C 180,E1 -10748.105,E2 -10748.105} C_VEL
LIN {X 0,Y 347.003,Z 515.36,A -85,B 0,C 180,E1 -10751.559,E2 -10751.559} C_VEL
LIN {X 0,Y 346.389,Z 508.952,A -85,B 0,C 180,E1 -10751.864,E2 -10751.864} C_VEL
LIN {X 0,Y 348.086,Z 481.6,A -85,B 0,C 180,E1 -10754.101,E2 -10754.101} C_VEL
LIN {X 0,Y 347.287,Z 481.364,A -85,B 0,C 180,E1 -10754.31,E2 -10754.31} C_VEL
LIN {X 0,Y 347.863,Z 483.611,A -85,B 0,C 180,E1 -10754.709,E2 -10754.709} C_VEL
LIN {X 0,Y 341.096,Z 525.415,A -85,B 0,C 180,E1 -10759.18,E2 -10759.18} C_VEL
LIN {X 0,Y 334.671,Z 569.319,A -85,B 0,C 180,E1 -10763.839,E2 -10763.839} C_VEL
LIN {X 0,Y 328.995,Z 613.752,A -85,B 0,C 180,E1 -10768.49,E2 -10768.49} C_VEL
LIN {X 0,Y 329.401,Z 624.04,A -85,B 0,C 180,E1 -10768.947,E2 -10768.947} C_VEL
LIN {X 0,Y 320.789,Z 743.675,A -85,B 0,C 180,E1 -10773.081,E2 -10773.081} C_VEL
LIN {X 0,Y 319.523,Z 769.481,A -85,B 0,C 180,E1 -10774.161,E2 -10774.161} C_VEL
LIN {X 0,Y 318.343,Z 786.464,A -85,B 0,C 180,E1 -10775.209,E2 -10775.209} C_VEL
LIN {X 0,Y 316.837,Z 802.926,A -85,B 0,C 180,E1 -10776.57,E2 -10776.57} C_VEL
LIN {X 0,Y 315.139,Z 818.215,A -85,B 0,C 180,E1 -10778.209,E2 -10778.209} C_VEL
LIN {X 0,Y 313.381,Z 832.59,A -85,B 0,C 180,E1 -10780.135,E2 -10780.135} C_VEL
LIN {X 0,Y 311.495,Z 846.867,A -85,B 0,C 180,E1 -10782.534,E2 -10782.534} C_VEL
LIN {X 0,Y 309.913,Z 858.762,A -85,B 0,C 180,E1 -10785.042,E2 -10785.042} C_VEL
LIN {X 0,Y 308.668,Z 868.784,A -85,B 0,C 180,E1 -10787.655,E2 -10787.655} C_VEL
LIN {X 0,Y 307.677,Z 877.805,A -85,B 0,C 180,E1 -10790.648,E2 -10790.648} C_VEL
LIN {X 0,Y 307.139,Z 884.278,A -85,B 0,C 180,E1 -10793.457,E2 -10793.457} C_VEL
LIN {X 0,Y 306.952,Z 889.642,A -85,B 0,C 180,E1 -10796.638,E2 -10796.638} C_VEL
LIN {X 0,Y 307.141,Z 893.018,A -85,B 0,C 180,E1 -10799.813,E2 -10799.813} C_VEL
LIN {X 0,Y 307.665,Z 894.558,A -85,B 0,C 180,E1 -10802.794,E2 -10802.794} C_VEL
LIN {X 0,Y 308.728,Z 894.327,A -85,B 0,C 180,E1 -10806.135,E2 -10806.135} C_VEL
LIN {X 0,Y 310.26,Z 892.257,A -85,B 0,C 180,E1 -10809.272,E2 -10809.272} C_VEL
LIN {X 0,Y 312.285,Z 888.663,A -85,B 0,C 180,E1 -10812.199,E2 -10812.199} C_VEL
LIN {X 0,Y 315.04,Z 882.95,A -85,B 0,C 180,E1 -10815.273,E2 -10815.273} C_VEL
LIN {X 0,Y 318.499,Z 875.103,A -85,B 0,C 180,E1 -10818.296,E2 -10818.296} C_VEL
LIN {X 0,Y 322.44,Z 865.514,A -85,B 0,C 180,E1 -10821.082,E2 -10821.082} C_VEL
LIN {X 0,Y 326.762,Z 854.277,A -85,B 0,C 180,E1 -10823.631,E2 -10823.631} C_VEL
LIN {X 0,Y 331.431,Z 841.289,A -85,B 0,C 180,E1 -10825.971,E2 -10825.971} C_VEL
LIN {X 0,Y 336.24,Z 827.076,A -85,B 0,C 180,E1 -10828.023,E2 -10828.023} C_VEL
LIN {X 0,Y 341.652,Z 810.792,A -85,B 0,C 180,E1 -10829.932,E2 -10829.932} C_VEL
LIN {X 0,Y 349.114,Z 790.021,A -85,B 0,C 180,E1 -10831.897,E2 -10831.897} C_VEL
LIN {X 0,Y 359.406,Z 765.647,A -85,B 0,C 180,E1 -10833.806,E2 -10833.806} C_VEL
LIN {X 0,Y 370.666,Z 738.791,A -85,B 0,C 180,E1 -10835.448,E2 -10835.448} C_VEL
LIN {X 0,Y 380.885,Z 711.451,A -85,B 0,C 180,E1 -10836.822,E2 -10836.822} C_VEL
LIN {X 0,Y 385.098,Z 698.612,A -85,B 0,C 180,E1 -10837.406,E2 -10837.406} C_VEL
LIN {X 0,Y 376.78,Z 726.758,A -85,B 0,C 180,E1 -10838.048,E2 -10838.048} C_VEL
LIN {X 0,Y 370.118,Z 747.925,A -85,B 0,C 180,E1 -10838.92,E2 -10838.92} C_VEL
LIN {X 0,Y 360.707,Z 776.463,A -85,B 0,C 180,E1 -10840.456,E2 -10840.456} C_VEL
LIN {X 0,Y 352.818,Z 799.622,A -85,B 0,C 180,E1 -10842.055,E2 -10842.055} C_VEL
LIN {X 0,Y 344.467,Z 824.415,A -85,B 0,C 180,E1 -10844.196,E2 -10844.196} C_VEL
LIN {X 0,Y 336.739,Z 848.042,A -85,B 0,C 180,E1 -10846.693,E2 -10846.693} C_VEL
LIN {X 0,Y 329.517,Z 870.936,A -85,B 0,C 180,E1 -10849.606,E2 -10849.606} C_VEL
LIN {X 0,Y 323.079,Z 892.392,A -85,B 0,C 180,E1 -10852.88,E2 -10852.88} C_VEL
LIN {X 0,Y 317.964,Z 910.667,A -85,B 0,C 180,E1 -10856.179,E2 -10856.179} C_VEL
LIN {X 0,Y 313.448,Z 928.224,A -85,B 0,C 180,E1 -10859.946,E2 -10859.946} C_VEL
LIN {X 0,Y 310.036,Z 943.159,A -85,B 0,C 180,E1 -10863.779,E2 -10863.779} C_VEL
LIN {X 0,Y 307.518,Z 956.251,A -85,B 0,C 180,E1 -10867.842,E2 -10867.842} C_VEL
LIN {X 0,Y 305.939,Z 966.894,A -85,B 0,C 180,E1 -10871.911,E2 -10871.911} C_VEL
LIN {X 0,Y 305.181,Z 974.557,A -85,B 0,C 180,E1 -10875.581,E2 -10875.581} C_VEL
LIN {X 0,Y 304.926,Z 980.523,A -85,B 0,C 180,E1 -10879.227,E2 -10879.227} C_VEL
LIN {X 0,Y 304.937,Z 984.749,A -85,B 0,C 180,E1 -10882.842,E2 -10882.842} C_VEL
LIN {X 0,Y 305.074,Z 987.276,A -85,B 0,C 180,E1 -10886.241,E2 -10886.241} C_VEL
LIN {X 0,Y 305.121,Z 988.32,A -85,B 0,C 180,E1 -10889.624,E2 -10889.624} C_VEL
LIN {X 0,Y 305.059,Z 987.889,A -85,B 0,C 180,E1 -10893.006,E2 -10893.006} C_VEL
LIN {X 0,Y 304.906,Z 985.953,A -85,B 0,C 180,E1 -10896.486,E2 -10896.486} C_VEL
LIN {X 0,Y 304.829,Z 982.388,A -85,B 0,C 180,E1 -10900.011,E2 -10900.011} C_VEL
LIN {X 0,Y 305.031,Z 977.117,A -85,B 0,C 180,E1 -10903.651,E2 -10903.651} C_VEL
LIN {X 0,Y 305.744,Z 969.638,A -85,B 0,C 180,E1 -10907.509,E2 -10907.509} C_VEL
LIN {X 0,Y 307.158,Z 960.056,A -85,B 0,C 180,E1 -10911.381,E2 -10911.381} C_VEL
LIN {X 0,Y 309.265,Z 948.826,A -85,B 0,C 180,E1 -10915.057,E2 -10915.057} C_VEL
LIN {X 0,Y 312.044,Z 936.048,A -85,B 0,C 180,E1 -10918.517,E2 -10918.517} C_VEL
LIN {X 0,Y 315.435,Z 921.786,A -85,B 0,C 180,E1 -10921.747,E2 -10921.747} C_VEL
LIN {X 0,Y 319.334,Z 906.053,A -85,B 0,C 180,E1 -10924.74,E2 -10924.74} C_VEL
LIN {X 0,Y 323.614,Z 888.87,A -85,B 0,C 180,E1 -10927.492,E2 -10927.492} C_VEL
LIN {X 0,Y 328.037,Z 870.847,A -85,B 0,C 180,E1 -10929.911,E2 -10929.911} C_VEL
LIN {X 0,Y 332.815,Z 850.674,A -85,B 0,C 180,E1 -10932.178,E2 -10932.178} C_VEL
LIN {X 0,Y 337.277,Z 830.755,A -85,B 0,C 180,E1 -10934.041,E2 -10934.041} C_VEL
LIN {X 0,Y 341.703,Z 809.219,A -85,B 0,C 180,E1 -10935.678,E2 -10935.678} C_VEL
LIN {X 0,Y 345.62,Z 787.675,A -85,B 0,C 180,E1 -10936.986,E2 -10936.986} C_VEL
LIN {X 0,Y 349.376,Z 763.836,A -85,B 0,C 180,E1 -10938.1,E2 -10938.1} C_VEL
LIN {X 0,Y 352.046,Z 741.199,A -85,B 0,C 180,E1 -10938.896,E2 -10938.896} C_VEL
LIN {X 0,Y 354.336,Z 716.702,A -85,B 0,C 180,E1 -10939.513,E2 -10939.513} C_VEL
LIN {X 0,Y 356.308,Z 702.739,A -85,B 0,C 180,E1 -10939.753,E2 -10939.753} C_VEL
LIN {X 0,Y 368.649,Z 673.453,A -85,B 0,C 180,E1 -10941.238,E2 -10941.238} C_VEL
LIN {X 0,Y 378.837,Z 652.441,A -85,B 0,C 180,E1 -10942.105,E2 -10942.105} C_VEL
LIN {X 0,Y 387.292,Z 636.16,A -85,B 0,C 180,E1 -10942.669,E2 -10942.669} C_VEL
LIN {X 0,Y 380.924,Z 618.583,A -85,B 0,C 180,E1 -10945.279,E2 -10945.279} C_VEL
LIN {X 0,Y 376.889,Z 600.399,A -85,B 0,C 180,E1 -10947.776,E2 -10947.776} C_VEL
LIN {X 0,Y 374.896,Z 580.738,A -85,B 0,C 180,E1 -10950.26,E2 -10950.26} C_VEL
LIN {X 0,Y 375.063,Z 558.746,A -85,B 0,C 180,E1 -10952.794,E2 -10952.794} C_VEL
LIN {X 0,Y 377.283,Z 536.758,A -85,B 0,C 180,E1 -10955.079,E2 -10955.079} C_VEL
LIN {X 0,Y 379.627,Z 522.518,A -85,B 0,C 180,E1 -10956.427,E2 -10956.427} C_VEL
LIN {X 0,Y 370.59,Z 504.937,A -85,B 0,C 180,E1 -10960.455,E2 -10960.455} C_VEL
LIN {X 0,Y 362.742,Z 490.351,A -85,B 0,C 180,E1 -10964.165,E2 -10964.165} C_VEL
LIN {X 0,Y 355.853,Z 477.719,A -85,B 0,C 180,E1 -10967.671,E2 -10967.671} C_VEL
LIN {X 0,Y 348.591,Z 464.772,A -85,B 0,C 180,E1 -10971.589,E2 -10971.589} C_VEL
LIN {X 0,Y 342.066,Z 453.491,A -85,B 0,C 180,E1 -10975.369,E2 -10975.369} C_VEL
LIN {X 0,Y 337.06,Z 444.778,A -85,B 0,C 180,E1 -10978.471,E2 -10978.471} C_VEL
LIN {X 0,Y 331.667,Z 435.343,A -85,B 0,C 180,E1 -10982.074,E2 -10982.074} C_VEL
LIN {X 0,Y 327.749,Z 429.115,A -85,B 0,C 180,E1 -10984.725,E2 -10984.725} C_VEL
LIN {X 0,Y 325.042,Z 424.409,A -85,B 0,C 180,E1 -10986.713,E2 -10986.713} C_VEL
LIN {X 0,Y 321.838,Z 419.107,A -85,B 0,C 180,E1 -10989.117,E2 -10989.117} C_VEL
LIN {X 0,Y 318.742,Z 413.878,A -85,B 0,C 180,E1 -10991.582,E2 -10991.582} C_VEL
LIN {X 0,Y 316.366,Z 409.945,A -85,B 0,C 180,E1 -10993.526,E2 -10993.526} C_VEL
LIN {X 0,Y 315.457,Z 408.435,A -85,B 0,C 180,E1 -10994.314,E2 -10994.314} C_VEL
LIN {X 0,Y 313.296,Z 404.988,A -85,B 0,C 180,E1 -10996.135,E2 -10996.135} C_VEL
LIN {X 0,Y 312.833,Z 403.64,A -85,B 0,C 180,E1 -10996.718,E2 -10996.718} C_VEL
LIN {X 0,Y 310.226,Z 400.298,A -85,B 0,C 180,E1 -10998.803,E2 -10998.803} C_VEL
LIN {X 0,Y 309.364,Z 397.999,A -85,B 0,C 180,E1 -10999.865,E2 -10999.865} C_VEL
LIN {X 0,Y 306.856,Z 394.813,A -85,B 0,C 180,E1 -11002.007,E2 -11002.007} C_VEL
LIN {X 0,Y 306.22,Z 392.586,A -85,B 0,C 180,E1 -11003.068,E2 -11003.068} C_VEL
LIN {X 0,Y 306.215,Z 392.662,A -85,B 0,C 180,E1 -11005.429,E2 -11005.429} C_VEL
LIN {X 0,Y 307.31,Z 395.746,A -85,B 0,C 180,E1 -11006.263,E2 -11006.263} C_VEL
LIN {X 0,Y 310.168,Z 398.727,A -85,B 0,C 180,E1 -11007.659,E2 -11007.659} C_VEL
LIN {X 0,Y 311.976,Z 402.338,A -85,B 0,C 180,E1 -11008.734,E2 -11008.734} C_VEL
LIN {X 0,Y 313.837,Z 404.49,A -85,B 0,C 180,E1 -11009.592,E2 -11009.592} C_VEL
LIN {X 0,Y 316.208,Z 408.518,A -85,B 0,C 180,E1 -11010.814,E2 -11010.814} C_VEL
LIN {X 0,Y 317.59,Z 410.815,A -85,B 0,C 180,E1 -11011.508,E2 -11011.508} C_VEL
LIN {X 0,Y 320.848,Z 416.1,A -85,B 0,C 180,E1 -11013.049,E2 -11013.049} C_VEL
LIN {X 0,Y 325.656,Z 424.288,A -85,B 0,C 180,E1 -11015.255,E2 -11015.255} C_VEL
LIN {X 0,Y 332.391,Z 437.182,A -85,B 0,C 180,E1 -11018.292,E2 -11018.292} C_VEL
LIN {X 0,Y 338.788,Z 451.132,A -85,B 0,C 180,E1 -11021.186,E2 -11021.186} C_VEL
LIN {X 0,Y 345.199,Z 467.142,A -85,B 0,C 180,E1 -11024.084,E2 -11024.084} C_VEL
LIN {X 0,Y 348.535,Z 476.678,A -85,B 0,C 180,E1 -11025.627,E2 -11025.627} C_VEL
LIN {X 0,Y 346.339,Z 510.029,A -85,B 0,C 180,E1 -11028.308,E2 -11028.308} C_VEL
LIN {X 0,Y 346.991,Z 517.921,A -85,B 0,C 180,E1 -11028.625,E2 -11028.625} C_VEL
LIN {X 0,Y 339.059,Z 710.11,A -85,B 0,C 180,E1 -11032.686,E2 -11032.686} C_VEL
LIN {X 0,Y 338.312,Z 729.705,A -85,B 0,C 180,E1 -11033.312,E2 -11033.312} C_VEL
LIN {X 0,Y 336.872,Z 748.456,A -85,B 0,C 180,E1 -11034.218,E2 -11034.218} C_VEL
LIN {X 0,Y 334.725,Z 766.624,A -85,B 0,C 180,E1 -11035.421,E2 -11035.421} C_VEL
LIN {X 0,Y 332.077,Z 783.591,A -85,B 0,C 180,E1 -11036.874,E2 -11036.874} C_VEL
LIN {X 0,Y 329.249,Z 798.843,A -85,B 0,C 180,E1 -11038.512,E2 -11038.512} C_VEL
LIN {X 0,Y 325.949,Z 813.933,A -85,B 0,C 180,E1 -11040.506,E2 -11040.506} C_VEL
LIN {X 0,Y 322.628,Z 827.477,A -85,B 0,C 180,E1 -11042.699,E2 -11042.699} C_VEL
LIN {X 0,Y 319.282,Z 840.051,A -85,B 0,C 180,E1 -11045.189,E2 -11045.189} C_VEL
LIN {X 0,Y 316.071,Z 851.408,A -85,B 0,C 180,E1 -11047.954,E2 -11047.954} C_VEL
LIN {X 0,Y 313.164,Z 861.44,A -85,B 0,C 180,E1 -11050.995,E2 -11050.995} C_VEL
LIN {X 0,Y 310.811,Z 869.624,A -85,B 0,C 180,E1 -11054.131,E2 -11054.131} C_VEL
LIN {X 0,Y 308.923,Z 876.351,A -85,B 0,C 180,E1 -11057.476,E2 -11057.476} C_VEL
LIN {X 0,Y 307.639,Z 881.295,A -85,B 0,C 180,E1 -11060.837,E2 -11060.837} C_VEL
LIN {X 0,Y 306.838,Z 884.758,A -85,B 0,C 180,E1 -11064.39,E2 -11064.39} C_VEL
LIN {X 0,Y 306.45,Z 886.541,A -85,B 0,C 180,E1 -11067.944,E2 -11067.944} C_VEL
LIN {X 0,Y 306.414,Z 886.699,A -85,B 0,C 180,E1 -11071.496,E2 -11071.496} C_VEL
LIN {X 0,Y 306.743,Z 885.239,A -85,B 0,C 180,E1 -11075.05,E2 -11075.05} C_VEL
LIN {X 0,Y 307.489,Z 882.022,A -85,B 0,C 180,E1 -11078.69,E2 -11078.69} C_VEL
LIN {X 0,Y 308.724,Z 877.193,A -85,B 0,C 180,E1 -11082.153,E2 -11082.153} C_VEL
LIN {X 0,Y 310.526,Z 870.724,A -85,B 0,C 180,E1 -11085.501,E2 -11085.501} C_VEL
LIN {X 0,Y 312.801,Z 862.822,A -85,B 0,C 180,E1 -11088.642,E2 -11088.642} C_VEL
LIN {X 0,Y 315.498,Z 853.536,A -85,B 0,C 180,E1 -11091.57,E2 -11091.57} C_VEL
LIN {X 0,Y 318.539,Z 842.898,A -85,B 0,C 180,E1 -11094.28,E2 -11094.28} C_VEL
LIN {X 0,Y 321.786,Z 830.903,A -85,B 0,C 180,E1 -11096.779,E2 -11096.779} C_VEL
LIN {X 0,Y 324.528,Z 820.124,A -85,B 0,C 180,E1 -11098.655,E2 -11098.655} C_VEL
LIN {X 0,Y 325.071,Z 814.646,A -85,B 0,C 180,E1 -11099.622,E2 -11099.622} C_VEL
LIN {X 0,Y 323.314,Z 801.45,A -85,B 0,C 180,E1 -11102.022,E2 -11102.022} C_VEL
LIN {X 0,Y 323.557,Z 795.384,A -85,B 0,C 180,E1 -11102.875,E2 -11102.875} C_VEL
LIN {X 0,Y 323.723,Z 794.454,A -85,B 0,C 180,E1 -11102.982,E2 -11102.982} C_VEL
LIN {X 0,Y 326.666,Z 778.35,A -85,B 0,C 180,E1 -11104.596,E2 -11104.596} C_VEL
LIN {X 0,Y 329.106,Z 761.937,A -85,B 0,C 180,E1 -11105.899,E2 -11105.899} C_VEL
LIN {X 0,Y 331.087,Z 743.811,A -85,B 0,C 180,E1 -11107.007,E2 -11107.007} C_VEL
LIN {X 0,Y 332.361,Z 725.394,A -85,B 0,C 180,E1 -11107.818,E2 -11107.818} C_VEL
LIN {X 0,Y 333.049,Z 702.745,A -85,B 0,C 180,E1 -11108.453,E2 -11108.453} C_VEL
LIN {X 0,Y 341.091,Z 516.617,A -85,B 0,C 180,E1 -11112.441,E2 -11112.441} C_VEL
LIN {X 0,Y 340.499,Z 509.999,A -85,B 0,C 180,E1 -11112.767,E2 -11112.767} C_VEL
LIN {X 0,Y 341.732,Z 490.957,A -85,B 0,C 180,E1 -11114.326,E2 -11114.326} C_VEL
LIN {X 0,Y 340.637,Z 491.152,A -85,B 0,C 180,E1 -11114.55,E2 -11114.55} C_VEL
LIN {X 0,Y 333.651,Z 533.081,A -85,B 0,C 180,E1 -11119.085,E2 -11119.085} C_VEL
LIN {X 0,Y 326.885,Z 578.162,A -85,B 0,C 180,E1 -11123.927,E2 -11123.927} C_VEL
LIN {X 0,Y 322.102,Z 614.735,A -85,B 0,C 180,E1 -11127.792,E2 -11127.792} C_VEL
LIN {X 0,Y 322.462,Z 624.903,A -85,B 0,C 180,E1 -11128.254,E2 -11128.254} C_VEL
LIN {X 0,Y 313.352,Z 745.736,A -85,B 0,C 180,E1 -11132.575,E2 -11132.575} C_VEL
LIN {X 0,Y 312.064,Z 770.719,A -85,B 0,C 180,E1 -11133.662,E2 -11133.662} C_VEL
LIN {X 0,Y 310.898,Z 786.719,A -85,B 0,C 180,E1 -11134.676,E2 -11134.676} C_VEL
LIN {X 0,Y 309.224,Z 804.208,A -85,B 0,C 180,E1 -11136.16,E2 -11136.16} C_VEL
LIN {X 0,Y 307.376,Z 820.193,A -85,B 0,C 180,E1 -11137.931,E2 -11137.931} C_VEL
LIN {X 0,Y 305.563,Z 834.412,A -85,B 0,C 180,E1 -11139.906,E2 -11139.906} C_VEL
LIN {X 0,Y 303.676,Z 848.282,A -85,B 0,C 180,E1 -11142.302,E2 -11142.302} C_VEL
LIN {X 0,Y 302.068,Z 860.039,A -85,B 0,C 180,E1 -11144.841,E2 -11144.841} C_VEL
LIN {X 0,Y 300.779,Z 870.062,A -85,B 0,C 180,E1 -11147.521,E2 -11147.521} C_VEL
LIN {X 0,Y 299.762,Z 879.098,A -85,B 0,C 180,E1 -11150.593,E2 -11150.593} C_VEL
LIN {X 0,Y 299.219,Z 885.628,A -85,B 0,C 180,E1 -11153.476,E2 -11153.476} C_VEL
LIN {X 0,Y 299.046,Z 891.056,A -85,B 0,C 180,E1 -11156.741,E2 -11156.741} C_VEL
LIN {X 0,Y 299.277,Z 894.482,A -85,B 0,C 180,E1 -11159.999,E2 -11159.999} C_VEL
LIN {X 0,Y 299.863,Z 896.099,A -85,B 0,C 180,E1 -11163.058,E2 -11163.058} C_VEL
LIN {X 0,Y 301.03,Z 895.959,A -85,B 0,C 180,E1 -11166.484,E2 -11166.484} C_VEL
LIN {X 0,Y 302.711,Z 893.989,A -85,B 0,C 180,E1 -11169.697,E2 -11169.697} C_VEL
LIN {X 0,Y 305.06,Z 890.245,A -85,B 0,C 180,E1 -11172.877,E2 -11172.877} C_VEL
LIN {X 0,Y 308.077,Z 884.602,A -85,B 0,C 180,E1 -11176.013,E2 -11176.013} C_VEL
LIN {X 0,Y 311.843,Z 876.855,A -85,B 0,C 180,E1 -11179.089,E2 -11179.089} C_VEL
LIN {X 0,Y 316.105,Z 867.441,A -85,B 0,C 180,E1 -11181.915,E2 -11181.915} C_VEL
LIN {X 0,Y 321.097,Z 855.658,A -85,B 0,C 180,E1 -11184.661,E2 -11184.661} C_VEL
LIN {X 0,Y 326.502,Z 842.134,A -85,B 0,C 180,E1 -11187.147,E2 -11187.147} C_VEL
LIN {X 0,Y 332.329,Z 827.007,A -85,B 0,C 180,E1 -11189.367,E2 -11189.367} C_VEL
LIN {X 0,Y 339.148,Z 809.101,A -85,B 0,C 180,E1 -11191.454,E2 -11191.454} C_VEL
LIN {X 0,Y 348.321,Z 788.122,A -85,B 0,C 180,E1 -11193.444,E2 -11193.444} C_VEL
LIN {X 0,Y 359.917,Z 763.661,A -85,B 0,C 180,E1 -11195.297,E2 -11195.297} C_VEL
LIN {X 0,Y 371.444,Z 738.039,A -85,B 0,C 180,E1 -11196.793,E2 -11196.793} C_VEL
LIN {X 0,Y 373.456,Z 733.241,A -85,B 0,C 180,E1 -11197.041,E2 -11197.041} C_VEL
LIN {X 0,Y 363.439,Z 761.464,A -85,B 0,C 180,E1 -11198.365,E2 -11198.365} C_VEL
LIN {X 0,Y 353.933,Z 786.929,A -85,B 0,C 180,E1 -11199.915,E2 -11199.915} C_VEL
LIN {X 0,Y 344.645,Z 811.667,A -85,B 0,C 180,E1 -11201.855,E2 -11201.855} C_VEL
LIN {X 0,Y 335.94,Z 835.269,A -85,B 0,C 180,E1 -11204.168,E2 -11204.168} C_VEL
LIN {X 0,Y 327.108,Z 860.164,A -85,B 0,C 180,E1 -11207.147,E2 -11207.147} C_VEL
LIN {X 0,Y 319.487,Z 882.756,A -85,B 0,C 180,E1 -11210.441,E2 -11210.441} C_VEL
LIN {X 0,Y 313.277,Z 902.383,A -85,B 0,C 180,E1 -11213.849,E2 -11213.849} C_VEL
LIN {X 0,Y 308.039,Z 920.348,A -85,B 0,C 180,E1 -11217.556,E2 -11217.556} C_VEL
LIN {X 0,Y 303.835,Z 936.371,A -85,B 0,C 180,E1 -11221.499,E2 -11221.499} C_VEL
LIN {X 0,Y 300.81,Z 949.75,A -85,B 0,C 180,E1 -11225.449,E2 -11225.449} C_VEL
LIN {X 0,Y 298.702,Z 961.29,A -85,B 0,C 180,E1 -11229.594,E2 -11229.594} C_VEL
LIN {X 0,Y 297.581,Z 969.895,A -85,B 0,C 180,E1 -11233.405,E2 -11233.405} C_VEL
LIN {X 0,Y 297.04,Z 976.989,A -85,B 0,C 180,E1 -11237.361,E2 -11237.361} C_VEL
LIN {X 0,Y 296.959,Z 981.926,A -85,B 0,C 180,E1 -11241.09,E2 -11241.09} C_VEL
LIN {X 0,Y 297.098,Z 985.257,A -85,B 0,C 180,E1 -11244.786,E2 -11244.786} C_VEL
LIN {X 0,Y 297.211,Z 986.847,A -85,B 0,C 180,E1 -11248.264,E2 -11248.264} C_VEL
LIN {X 0,Y 297.199,Z 986.979,A -85,B 0,C 180,E1 -11251.735,E2 -11251.735} C_VEL
LIN {X 0,Y 297.055,Z 985.615,A -85,B 0,C 180,E1 -11255.214,E2 -11255.214} C_VEL
LIN {X 0,Y 296.908,Z 982.534,A -85,B 0,C 180,E1 -11258.911,E2 -11258.911} C_VEL
LIN {X 0,Y 296.982,Z 978.008,A -85,B 0,C 180,E1 -11262.488,E2 -11262.488} C_VEL
LIN {X 0,Y 297.517,Z 971.272,A -85,B 0,C 180,E1 -11266.397,E2 -11266.397} C_VEL
LIN {X 0,Y 298.732,Z 962.273,A -85,B 0,C 180,E1 -11270.421,E2 -11270.421} C_VEL
LIN {X 0,Y 300.624,Z 951.875,A -85,B 0,C 180,E1 -11274.147,E2 -11274.147} C_VEL
LIN {X 0,Y 303.23,Z 939.84,A -85,B 0,C 180,E1 -11277.705,E2 -11277.705} C_VEL
LIN {X 0,Y 306.457,Z 926.39,A -85,B 0,C 180,E1 -11281.03,E2 -11281.03} C_VEL
LIN {X 0,Y 310.459,Z 910.565,A -85,B 0,C 180,E1 -11284.305,E2 -11284.305} C_VEL
LIN {X 0,Y 314.838,Z 893.634,A -85,B 0,C 180,E1 -11287.227,E2 -11287.227} C_VEL
LIN {X 0,Y 319.385,Z 875.832,A -85,B 0,C 180,E1 -11289.806,E2 -11289.806} C_VEL
LIN {X 0,Y 324.148,Z 856.618,A -85,B 0,C 180,E1 -11292.136,E2 -11292.136} C_VEL
LIN {X 0,Y 328.85,Z 836.636,A -85,B 0,C 180,E1 -11294.148,E2 -11294.148} C_VEL
LIN {X 0,Y 333.588,Z 814.964,A -85,B 0,C 180,E1 -11295.944,E2 -11295.944} C_VEL
LIN {X 0,Y 337.887,Z 793.208,A -85,B 0,C 180,E1 -11297.392,E2 -11297.392} C_VEL
LIN {X 0,Y 341.795,Z 770.387,A -85,B 0,C 180,E1 -11298.567,E2 -11298.567} C_VEL
LIN {X 0,Y 344.867,Z 747.671,A -85,B 0,C 180,E1 -11299.451,E2 -11299.451} C_VEL
LIN {X 0,Y 347.476,Z 720.535,A -85,B 0,C 180,E1 -11300.216,E2 -11300.216} C_VEL
LIN {X 0,Y 350.154,Z 701.818,A -85,B 0,C 180,E1 -11300.57,E2 -11300.57} C_VEL
LIN {X 0,Y 362.616,Z 672.692,A -85,B 0,C 180,E1 -11302.054,E2 -11302.054} C_VEL
LIN {X 0,Y 372.851,Z 651.68,A -85,B 0,C 180,E1 -11302.919,E2 -11302.919} C_VEL
LIN {X 0,Y 379.984,Z 638.103,A -85,B 0,C 180,E1 -11303.392,E2 -11303.392} C_VEL
LIN {X 0,Y 374.184,Z 621.075,A -85,B 0,C 180,E1 -11305.929,E2 -11305.929} C_VEL
LIN {X 0,Y 370.452,Z 603.028,A -85,B 0,C 180,E1 -11308.426,E2 -11308.426} C_VEL
LIN {X 0,Y 368.685,Z 583.19,A -85,B 0,C 180,E1 -11310.959,E2 -11310.959} C_VEL
LIN {X 0,Y 369.031,Z 561,A -85,B 0,C 180,E1 -11313.532,E2 -11313.532} C_VEL
LIN {X 0,Y 371.55,Z 538.021,A -85,B 0,C 180,E1 -11315.932,E2 -11315.932} C_VEL
LIN {X 0,Y 373.369,Z 526.479,A -85,B 0,C 180,E1 -11317.068,E2 -11317.068} C_VEL
LIN {X 0,Y 364.466,Z 509.121,A -85,B 0,C 180,E1 -11321.113,E2 -11321.113} C_VEL
LIN {X 0,Y 356.71,Z 494.495,A -85,B 0,C 180,E1 -11324.89,E2 -11324.89} C_VEL
LIN {X 0,Y 348.911,Z 480.249,A -85,B 0,C 180,E1 -11328.931,E2 -11328.931} C_VEL
LIN {X 0,Y 340.87,Z 465.981,A -85,B 0,C 180,E1 -11333.432,E2 -11333.432} C_VEL
LIN {X 0,Y 334.804,Z 455.494,A -85,B 0,C 180,E1 -11337.09,E2 -11337.09} C_VEL
LIN {X 0,Y 329.197,Z 445.812,A -85,B 0,C 180,E1 -11340.697,E2 -11340.697} C_VEL
LIN {X 0,Y 325.773,Z 440.125,A -85,B 0,C 180,E1 -11342.991,E2 -11342.991} C_VEL
LIN {X 0,Y 322.978,Z 435.389,A -85,B 0,C 180,E1 -11344.973,E2 -11344.973} C_VEL
LIN {X 0,Y 320.001,Z 430.309,A -85,B 0,C 180,E1 -11347.18,E2 -11347.18} C_VEL
LIN {X 0,Y 317.184,Z 425.481,A -85,B 0,C 180,E1 -11349.368,E2 -11349.368} C_VEL
LIN {X 0,Y 314.231,Z 420.421,A -85,B 0,C 180,E1 -11351.751,E2 -11351.751} C_VEL
LIN {X 0,Y 311.624,Z 416.008,A -85,B 0,C 180,E1 -11353.925,E2 -11353.925} C_VEL
LIN {X 0,Y 308.636,Z 411.214,A -85,B 0,C 180,E1 -11356.481,E2 -11356.481} C_VEL
LIN {X 0,Y 307.789,Z 409.744,A -85,B 0,C 180,E1 -11357.243,E2 -11357.243} C_VEL
LIN {X 0,Y 305.352,Z 405.949,A -85,B 0,C 180,E1 -11359.433,E2 -11359.433} C_VEL
LIN {X 0,Y 304.67,Z 404.426,A -85,B 0,C 180,E1 -11360.186,E2 -11360.186} C_VEL
LIN {X 0,Y 302.25,Z 401.082,A -85,B 0,C 180,E1 -11362.361,E2 -11362.361} C_VEL
LIN {X 0,Y 301.372,Z 398.945,A -85,B 0,C 180,E1 -11363.461,E2 -11363.461} C_VEL
LIN {X 0,Y 300.672,Z 398.343,A -85,B 0,C 180,E1 -11364.144,E2 -11364.144} C_VEL
LIN {X 0,Y 302.423,Z 399.864,A -85,B 0,C 180,E1 -11365.058,E2 -11365.058} C_VEL
LIN {X 0,Y 304.368,Z 403.64,A -85,B 0,C 180,E1 -11366.327,E2 -11366.327} C_VEL
LIN {X 0,Y 306.192,Z 405.345,A -85,B 0,C 180,E1 -11367.205,E2 -11367.205} C_VEL
LIN {X 0,Y 308.44,Z 409.486,A -85,B 0,C 180,E1 -11368.54,E2 -11368.54} C_VEL
LIN {X 0,Y 309.735,Z 411.038,A -85,B 0,C 180,E1 -11369.173,E2 -11369.173} C_VEL
LIN {X 0,Y 312.475,Z 415.487,A -85,B 0,C 180,E1 -11370.582,E2 -11370.582} C_VEL
LIN {X 0,Y 318.805,Z 426.251,A -85,B 0,C 180,E1 -11373.72,E2 -11373.72} C_VEL
LIN {X 0,Y 325.328,Z 438.528,A -85,B 0,C 180,E1 -11376.821,E2 -11376.821} C_VEL
LIN {X 0,Y 331.607,Z 451.79,A -85,B 0,C 180,E1 -11379.748,E2 -11379.748} C_VEL
LIN {X 0,Y 337.842,Z 467.056,A -85,B 0,C 180,E1 -11382.668,E2 -11382.668} C_VEL
LIN {X 0,Y 342.583,Z 480.22,A -85,B 0,C 180,E1 -11384.906,E2 -11384.906} C_VEL
LIN {X 0,Y 340.459,Z 511.459,A -85,B 0,C 180,E1 -11387.429,E2 -11387.429} C_VEL
LIN {X 0,Y 341.058,Z 519.195,A -85,B 0,C 180,E1 -11387.744,E2 -11387.744} C_VEL
LIN {X 0,Y 332.795,Z 710.659,A -85,B 0,C 180,E1 -11391.843,E2 -11391.843} C_VEL
LIN {X 0,Y 332.025,Z 730.306,A -85,B 0,C 180,E1 -11392.473,E2 -11392.473} C_VEL
LIN {X 0,Y 330.57,Z 748.778,A -85,B 0,C 180,E1 -11393.366,E2 -11393.366} C_VEL
LIN {X 0,Y 328.416,Z 766.759,A -85,B 0,C 180,E1 -11394.552,E2 -11394.552} C_VEL
LIN {X 0,Y 325.651,Z 783.979,A -85,B 0,C 180,E1 -11396.028,E2 -11396.028} C_VEL
LIN {X 0,Y 322.536,Z 800.097,A -85,B 0,C 180,E1 -11397.779,E2 -11397.779} C_VEL
LIN {X 0,Y 319.092,Z 815.19,A -85,B 0,C 180,E1 -11399.807,E2 -11399.807} C_VEL
LIN {X 0,Y 315.62,Z 828.738,A -85,B 0,C 180,E1 -11402.041,E2 -11402.041} C_VEL
LIN {X 0,Y 312.114,Z 841.314,A -85,B 0,C 180,E1 -11404.579,E2 -11404.579} C_VEL
LIN {X 0,Y 308.815,Z 852.445,A -85,B 0,C 180,E1 -11407.339,E2 -11407.339} C_VEL
LIN {X 0,Y 305.849,Z 862.168,A -85,B 0,C 180,E1 -11410.323,E2 -11410.323} C_VEL
LIN {X 0,Y 303.197,Z 870.891,A -85,B 0,C 180,E1 -11413.722,E2 -11413.722} C_VEL
LIN {X 0,Y 301.195,Z 877.618,A -85,B 0,C 180,E1 -11417.15,E2 -11417.15} C_VEL
LIN {X 0,Y 299.826,Z 882.561,A -85,B 0,C 180,E1 -11420.596,E2 -11420.596} C_VEL
LIN {X 0,Y 298.969,Z 886.023,A -85,B 0,C 180,E1 -11424.242,E2 -11424.242} C_VEL
LIN {X 0,Y 298.554,Z 887.804,A -85,B 0,C 180,E1 -11427.889,E2 -11427.889} C_VEL
LIN {X 0,Y 298.517,Z 887.963,A -85,B 0,C 180,E1 -11431.536,E2 -11431.536} C_VEL
LIN {X 0,Y 298.868,Z 886.502,A -85,B 0,C 180,E1 -11435.183,E2 -11435.183} C_VEL
LIN {X 0,Y 299.641,Z 883.381,A -85,B 0,C 180,E1 -11438.83,E2 -11438.83} C_VEL
LIN {X 0,Y 300.983,Z 878.457,A -85,B 0,C 180,E1 -11442.471,E2 -11442.471} C_VEL
LIN {X 0,Y 302.896,Z 871.989,A -85,B 0,C 180,E1 -11445.902,E2 -11445.902} C_VEL
LIN {X 0,Y 305.301,Z 864.085,A -85,B 0,C 180,E1 -11449.118,E2 -11449.118} C_VEL
LIN {X 0,Y 308.143,Z 854.796,A -85,B 0,C 180,E1 -11452.111,E2 -11452.111} C_VEL
LIN {X 0,Y 311.338,Z 844.156,A -85,B 0,C 180,E1 -11454.88,E2 -11454.88} C_VEL
LIN {X 0,Y 314.741,Z 832.158,A -85,B 0,C 180,E1 -11457.428,E2 -11457.428} C_VEL
LIN {X 0,Y 318.273,Z 818.718,A -85,B 0,C 180,E1 -11459.76,E2 -11459.76} C_VEL
LIN {X 0,Y 321.661,Z 804.362,A -85,B 0,C 180,E1 -11461.795,E2 -11461.795} C_VEL
LIN {X 0,Y 323.723,Z 794.454,A -85,B 0,C 180,E1 -11462.982,E2 -11462.982} C_VEL
LIN {X 0,Y 324.172,Z 788.138,A -85,B 0,C 180,E1 -11463.778,E2 -11463.778} C_VEL
LIN {X 0,Y 322.28,Z 773.13,A -85,B 0,C 180,E1 -11465.819,E2 -11465.819} C_VEL
LIN {X 0,Y 322.33,Z 766.359,A -85,B 0,C 180,E1 -11466.487,E2 -11466.487} C_VEL
LIN {X 0,Y 322.437,Z 765.346,A -85,B 0,C 180,E1 -11466.564,E2 -11466.564} C_VEL
LIN {X 0,Y 324.59,Z 747.178,A -85,B 0,C 180,E1 -11467.73,E2 -11467.73} C_VEL
LIN {X 0,Y 326.045,Z 728.082,A -85,B 0,C 180,E1 -11468.614,E2 -11468.614} C_VEL
LIN {X 0,Y 326.794,Z 706.538,A -85,B 0,C 180,E1 -11469.254,E2 -11469.254} C_VEL
LIN {X 0,Y 335.261,Z 517.887,A -85,B 0,C 180,E1 -11473.353,E2 -11473.353} C_VEL
LIN {X 0,Y 334.705,Z 511.054,A -85,B 0,C 180,E1 -11473.703,E2 -11473.703} C_VEL
LIN {X 0,Y 335.186,Z 502.595,A -85,B 0,C 180,E1 -11474.403,E2 -11474.403} C_VEL
LIN {X 0,Y 332.581,Z 503.086,A -85,B 0,C 180,E1 -11474.866,E2 -11474.866} C_VEL
LIN {X 0,Y 325.433,Z 545.202,A -85,B 0,C 180,E1 -11479.472,E2 -11479.472} C_VEL
LIN {X 0,Y 318.576,Z 590.379,A -85,B 0,C 180,E1 -11484.379,E2 -11484.379} C_VEL
LIN {X 0,Y 315.223,Z 615.677,A -85,B 0,C 180,E1 -11487.071,E2 -11487.071} C_VEL
LIN {X 0,Y 315.539,Z 625.657,A -85,B 0,C 180,E1 -11487.54,E2 -11487.54} C_VEL
LIN {X 0,Y 306.506,Z 738.784,A -85,B 0,C 180,E1 -11491.69,E2 -11491.69} C_VEL
LIN {X 0,Y 304.68,Z 770.474,A -85,B 0,C 180,E1 -11493.078,E2 -11493.078} C_VEL
LIN {X 0,Y 303.357,Z 788.037,A -85,B 0,C 180,E1 -11494.21,E2 -11494.21} C_VEL
LIN {X 0,Y 301.625,Z 805.444,A -85,B 0,C 180,E1 -11495.729,E2 -11495.729} C_VEL
LIN {X 0,Y 299.732,Z 821.255,A -85,B 0,C 180,E1 -11497.524,E2 -11497.524} C_VEL
LIN {X 0,Y 297.837,Z 835.612,A -85,B 0,C 180,E1 -11499.565,E2 -11499.565} C_VEL
LIN {X 0,Y 295.835,Z 849.778,A -85,B 0,C 180,E1 -11502.087,E2 -11502.087} C_VEL
LIN {X 0,Y 294.107,Z 862.006,A -85,B 0,C 180,E1 -11504.824,E2 -11504.824} C_VEL
LIN {X 0,Y 292.794,Z 871.981,A -85,B 0,C 180,E1 -11507.599,E2 -11507.599} C_VEL
LIN {X 0,Y 291.799,Z 880.906,A -85,B 0,C 180,E1 -11510.732,E2 -11510.732} C_VEL
LIN {X 0,Y 291.254,Z 887.704,A -85,B 0,C 180,E1 -11513.89,E2 -11513.89} C_VEL
LIN {X 0,Y 291.14,Z 892.706,A -85,B 0,C 180,E1 -11517.047,E2 -11517.047} C_VEL
LIN {X 0,Y 291.474,Z 896.276,A -85,B 0,C 180,E1 -11520.589,E2 -11520.589} C_VEL
LIN {X 0,Y 292.242,Z 897.745,A -85,B 0,C 180,E1 -11523.923,E2 -11523.923} C_VEL
LIN {X 0,Y 293.532,Z 897.483,A -85,B 0,C 180,E1 -11527.24,E2 -11527.24} C_VEL
LIN {X 0,Y 295.594,Z 895.285,A -85,B 0,C 180,E1 -11530.721,E2 -11530.721} C_VEL
LIN {X 0,Y 298.423,Z 891.046,A -85,B 0,C 180,E1 -11534.157,E2 -11534.157} C_VEL
LIN {X 0,Y 301.852,Z 885.097,A -85,B 0,C 180,E1 -11537.344,E2 -11537.344} C_VEL
LIN {X 0,Y 305.541,Z 878.159,A -85,B 0,C 180,E1 -11540.096,E2 -11540.096} C_VEL
LIN {X 0,Y 309.888,Z 869.503,A -85,B 0,C 180,E1 -11542.779,E2 -11542.779} C_VEL
LIN {X 0,Y 314.91,Z 858.873,A -85,B 0,C 180,E1 -11545.38,E2 -11545.38} C_VEL
LIN {X 0,Y 320.681,Z 846.073,A -85,B 0,C 180,E1 -11547.884,E2 -11547.884} C_VEL
LIN {X 0,Y 327.367,Z 830.849,A -85,B 0,C 180,E1 -11550.261,E2 -11550.261} C_VEL
LIN {X 0,Y 334.952,Z 813.626,A -85,B 0,C 180,E1 -11552.399,E2 -11552.399} C_VEL
LIN {X 0,Y 344.94,Z 793.332,A -85,B 0,C 180,E1 -11554.418,E2 -11554.418} C_VEL
LIN {X 0,Y 356.803,Z 770.844,A -85,B 0,C 180,E1 -11556.19,E2 -11556.19} C_VEL
LIN {X 0,Y 362.87,Z 758.954,A -85,B 0,C 180,E1 -11556.958,E2 -11556.958} C_VEL
LIN {X 0,Y 352.1,Z 785.219,A -85,B 0,C 180,E1 -11558.524,E2 -11558.524} C_VEL
LIN {X 0,Y 342.349,Z 808.65,A -85,B 0,C 180,E1 -11560.334,E2 -11560.334} C_VEL
LIN {X 0,Y 332.252,Z 833.251,A -85,B 0,C 180,E1 -11562.753,E2 -11562.753} C_VEL
LIN {X 0,Y 322.948,Z 856.836,A -85,B 0,C 180,E1 -11565.596,E2 -11565.596} C_VEL
LIN {X 0,Y 314.546,Z 879.213,A -85,B 0,C 180,E1 -11568.882,E2 -11568.882} C_VEL
LIN {X 0,Y 307.47,Z 899.383,A -85,B 0,C 180,E1 -11572.429,E2 -11572.429} C_VEL
LIN {X 0,Y 301.694,Z 917.273,A -85,B 0,C 180,E1 -11576.166,E2 -11576.166} C_VEL
LIN {X 0,Y 296.861,Z 933.917,A -85,B 0,C 180,E1 -11580.322,E2 -11580.322} C_VEL
LIN {X 0,Y 293.336,Z 948.011,A -85,B 0,C 180,E1 -11584.565,E2 -11584.565} C_VEL
LIN {X 0,Y 290.984,Z 959.685,A -85,B 0,C 180,E1 -11588.85,E2 -11588.85} C_VEL
LIN {X 0,Y 289.677,Z 968.719,A -85,B 0,C 180,E1 -11592.958,E2 -11592.958} C_VEL
LIN {X 0,Y 289.097,Z 975.75,A -85,B 0,C 180,E1 -11597.008,E2 -11597.008} C_VEL
LIN {X 0,Y 289.004,Z 980.704,A -85,B 0,C 180,E1 -11600.842,E2 -11600.842} C_VEL
LIN {X 0,Y 289.167,Z 983.895,A -85,B 0,C 180,E1 -11604.444,E2 -11604.444} C_VEL
LIN {X 0,Y 289.299,Z 985.549,A -85,B 0,C 180,E1 -11608.019,E2 -11608.019} C_VEL
LIN {X 0,Y 289.309,Z 985.759,A -85,B 0,C 180,E1 -11611.386,E2 -11611.386} C_VEL
LIN {X 0,Y 289.157,Z 984.523,A -85,B 0,C 180,E1 -11614.959,E2 -11614.959} C_VEL
LIN {X 0,Y 288.993,Z 981.527,A -85,B 0,C 180,E1 -11618.756,E2 -11618.756} C_VEL
LIN {X 0,Y 289.037,Z 977.155,A -85,B 0,C 180,E1 -11622.384,E2 -11622.384} C_VEL
LIN {X 0,Y 289.566,Z 970.39,A -85,B 0,C 180,E1 -11626.447,E2 -11626.447} C_VEL
LIN {X 0,Y 290.7,Z 962.045,A -85,B 0,C 180,E1 -11630.327,E2 -11630.327} C_VEL
LIN {X 0,Y 292.497,Z 952.294,A -85,B 0,C 180,E1 -11634.002,E2 -11634.002} C_VEL
LIN {X 0,Y 295.095,Z 940.529,A -85,B 0,C 180,E1 -11637.657,E2 -11637.657} C_VEL
LIN {X 0,Y 298.552,Z 926.48,A -85,B 0,C 180,E1 -11641.271,E2 -11641.271} C_VEL
LIN {X 0,Y 302.696,Z 910.59,A -85,B 0,C 180,E1 -11644.666,E2 -11644.666} C_VEL
LIN {X 0,Y 307.376,Z 893.098,A -85,B 0,C 180,E1 -11647.773,E2 -11647.773} C_VEL
LIN {X 0,Y 312.135,Z 875.057,A -85,B 0,C 180,E1 -11650.441,E2 -11650.441} C_VEL
LIN {X 0,Y 317.253,Z 855.04,A -85,B 0,C 180,E1 -11652.901,E2 -11652.901} C_VEL
LIN {X 0,Y 322.129,Z 834.827,A -85,B 0,C 180,E1 -11654.953,E2 -11654.953} C_VEL
LIN {X 0,Y 327.075,Z 812.805,A -85,B 0,C 180,E1 -11656.784,E2 -11656.784} C_VEL
LIN {X 0,Y 331.456,Z 791.126,A -85,B 0,C 180,E1 -11658.231,E2 -11658.231} C_VEL
LIN {X 0,Y 335.477,Z 768.273,A -85,B 0,C 180,E1 -11659.417,E2 -11659.417} C_VEL
LIN {X 0,Y 338.647,Z 745.024,A -85,B 0,C 180,E1 -11660.32,E2 -11660.32} C_VEL
LIN {X 0,Y 341.263,Z 719.044,A -85,B 0,C 180,E1 -11661.05,E2 -11661.05} C_VEL
LIN {X 0,Y 344.091,Z 700.594,A -85,B 0,C 180,E1 -11661.412,E2 -11661.412} C_VEL
LIN {X 0,Y 357.103,Z 670.744,A -85,B 0,C 180,E1 -11662.937,E2 -11662.937} C_VEL
LIN {X 0,Y 367.886,Z 649.148,A -85,B 0,C 180,E1 -11663.823,E2 -11663.823} C_VEL
LIN {X 0,Y 372.747,Z 640.017,A -85,B 0,C 180,E1 -11664.141,E2 -11664.141} C_VEL
LIN {X 0,Y 367.127,Z 622.088,A -85,B 0,C 180,E1 -11666.811,E2 -11666.811} C_VEL
LIN {X 0,Y 363.628,Z 602.44,A -85,B 0,C 180,E1 -11669.515,E2 -11669.515} C_VEL
LIN {X 0,Y 362.371,Z 581.872,A -85,B 0,C 180,E1 -11672.116,E2 -11672.116} C_VEL
LIN {X 0,Y 363.347,Z 558.98,A -85,B 0,C 180,E1 -11674.753,E2 -11674.753} C_VEL
LIN {X 0,Y 366.593,Z 535.143,A -85,B 0,C 180,E1 -11677.214,E2 -11677.214} C_VEL
LIN {X 0,Y 367.228,Z 530.628,A -85,B 0,C 180,E1 -11677.678,E2 -11677.678} C_VEL
LIN {X 0,Y 358.368,Z 513.248,A -85,B 0,C 180,E1 -11681.792,E2 -11681.792} C_VEL
LIN {X 0,Y 350.87,Z 499.245,A -85,B 0,C 180,E1 -11685.477,E2 -11685.477} C_VEL
LIN {X 0,Y 343.73,Z 486.021,A -85,B 0,C 180,E1 -11689.271,E2 -11689.271} C_VEL
LIN {X 0,Y 335.952,Z 472.12,A -85,B 0,C 180,E1 -11693.678,E2 -11693.678} C_VEL
LIN {X 0,Y 329.813,Z 461.508,A -85,B 0,C 180,E1 -11697.394,E2 -11697.394} C_VEL
LIN {X 0,Y 324.208,Z 451.779,A -85,B 0,C 180,E1 -11701.061,E2 -11701.061} C_VEL
LIN {X 0,Y 318.791,Z 442.431,A -85,B 0,C 180,E1 -11704.858,E2 -11704.858} C_VEL
LIN {X 0,Y 315.192,Z 436.517,A -85,B 0,C 180,E1 -11707.474,E2 -11707.474} C_VEL
LIN {X 0,Y 312.387,Z 431.716,A -85,B 0,C 180,E1 -11709.663,E2 -11709.663} C_VEL
LIN {X 0,Y 309.358,Z 426.571,A -85,B 0,C 180,E1 -11712.128,E2 -11712.128} C_VEL
LIN {X 0,Y 306.155,Z 421.223,A -85,B 0,C 180,E1 -11714.831,E2 -11714.831} C_VEL
LIN {X 0,Y 303.941,Z 417.419,A -85,B 0,C 180,E1 -11716.828,E2 -11716.828} C_VEL
LIN {X 0,Y 302.628,Z 415.57,A -85,B 0,C 180,E1 -11717.914,E2 -11717.914} C_VEL
LIN {X 0,Y 300.497,Z 411.588,A -85,B 0,C 180,E1 -11720.043,E2 -11720.043} C_VEL
LIN {X 0,Y 297.638,Z 407.336,A -85,B 0,C 180,E1 -11722.726,E2 -11722.726} C_VEL
LIN {X 0,Y 296.91,Z 405.526,A -85,B 0,C 180,E1 -11723.749,E2 -11723.749} C_VEL
LIN {X 0,Y 298.658,Z 406.69,A -85,B 0,C 180,E1 -11724.634,E2 -11724.634} C_VEL
LIN {X 0,Y 300.783,Z 410.615,A -85,B 0,C 180,E1 -11726.027,E2 -11726.027} C_VEL
LIN {X 0,Y 302.504,Z 412.575,A -85,B 0,C 180,E1 -11726.926,E2 -11726.926} C_VEL
LIN {X 0,Y 305.049,Z 416.743,A -85,B 0,C 180,E1 -11728.377,E2 -11728.377} C_VEL
LIN {X 0,Y 309.368,Z 423.896,A -85,B 0,C 180,E1 -11730.718,E2 -11730.718} C_VEL
LIN {X 0,Y 314.188,Z 432.09,A -85,B 0,C 180,E1 -11733.187,E2 -11733.187} C_VEL
LIN {X 0,Y 320.567,Z 444.369,A -85,B 0,C 180,E1 -11736.343,E2 -11736.343} C_VEL
LIN {X 0,Y 326.696,Z 457.601,A -85,B 0,C 180,E1 -11739.311,E2 -11739.311} C_VEL
LIN {X 0,Y 332.816,Z 473.02,A -85,B 0,C 180,E1 -11742.296,E2 -11742.296} C_VEL
LIN {X 0,Y 336.662,Z 484.218,A -85,B 0,C 180,E1 -11744.202,E2 -11744.202} C_VEL
LIN {X 0,Y 334.648,Z 512.763,A -85,B 0,C 180,E1 -11746.513,E2 -11746.513} C_VEL
LIN {X 0,Y 335.214,Z 520.342,A -85,B 0,C 180,E1 -11746.83,E2 -11746.83} C_VEL
LIN {X 0,Y 326.608,Z 711.065,A -85,B 0,C 180,E1 -11750.963,E2 -11750.963} C_VEL
LIN {X 0,Y 325.811,Z 730.908,A -85,B 0,C 180,E1 -11751.6,E2 -11751.6} C_VEL
LIN {X 0,Y 324.323,Z 749.289,A -85,B 0,C 180,E1 -11752.492,E2 -11752.492} C_VEL
LIN {X 0,Y 322.174,Z 766.784,A -85,B 0,C 180,E1 -11753.647,E2 -11753.647} C_VEL
LIN {X 0,Y 319.296,Z 784.334,A -85,B 0,C 180,E1 -11755.146,E2 -11755.146} C_VEL
LIN {X 0,Y 316.042,Z 800.648,A -85,B 0,C 180,E1 -11756.926,E2 -11756.926} C_VEL
LIN {X 0,Y 312.439,Z 815.867,A -85,B 0,C 180,E1 -11758.988,E2 -11758.988} C_VEL
LIN {X 0,Y 308.655,Z 829.998,A -85,B 0,C 180,E1 -11761.352,E2 -11761.352} C_VEL
LIN {X 0,Y 304.984,Z 842.577,A -85,B 0,C 180,E1 -11763.941,E2 -11763.941} C_VEL
LIN {X 0,Y 301.522,Z 853.71,A -85,B 0,C 180,E1 -11766.759,E2 -11766.759} C_VEL
LIN {X 0,Y 298.399,Z 863.434,A -85,B 0,C 180,E1 -11769.811,E2 -11769.811} C_VEL
LIN {X 0,Y 295.597,Z 872.158,A -85,B 0,C 180,E1 -11773.291,E2 -11773.291} C_VEL
LIN {X 0,Y 293.477,Z 878.885,A -85,B 0,C 180,E1 -11776.806,E2 -11776.806} C_VEL
LIN {X 0,Y 291.971,Z 884.01,A -85,B 0,C 180,E1 -11780.495,E2 -11780.495} C_VEL
LIN {X 0,Y 291.102,Z 887.288,A -85,B 0,C 180,E1 -11784.086,E2 -11784.086} C_VEL
LIN {X 0,Y 290.659,Z 889.068,A -85,B 0,C 180,E1 -11787.832,E2 -11787.832} C_VEL
LIN {X 0,Y 290.62,Z 889.226,A -85,B 0,C 180,E1 -11791.578,E2 -11791.578} C_VEL
LIN {X 0,Y 290.995,Z 887.766,A -85,B 0,C 180,E1 -11795.324,E2 -11795.324} C_VEL
LIN {X 0,Y 291.821,Z 884.646,A -85,B 0,C 180,E1 -11799.069,E2 -11799.069} C_VEL
LIN {X 0,Y 293.252,Z 879.722,A -85,B 0,C 180,E1 -11802.805,E2 -11802.805} C_VEL
LIN {X 0,Y 295.282,Z 873.253,A -85,B 0,C 180,E1 -11806.323,E2 -11806.323} C_VEL
LIN {X 0,Y 297.823,Z 865.348,A -85,B 0,C 180,E1 -11809.617,E2 -11809.617} C_VEL
LIN {X 0,Y 300.819,Z 856.057,A -85,B 0,C 180,E1 -11812.679,E2 -11812.679} C_VEL
LIN {X 0,Y 304.172,Z 845.414,A -85,B 0,C 180,E1 -11815.507,E2 -11815.507} C_VEL
LIN {X 0,Y 307.739,Z 833.412,A -85,B 0,C 180,E1 -11818.107,E2 -11818.107} C_VEL
LIN {X 0,Y 311.432,Z 819.967,A -85,B 0,C 180,E1 -11820.482,E2 -11820.482} C_VEL
LIN {X 0,Y 314.97,Z 805.606,A -85,B 0,C 180,E1 -11822.553,E2 -11822.553} C_VEL
LIN {X 0,Y 318.192,Z 790.44,A -85,B 0,C 180,E1 -11824.337,E2 -11824.337} C_VEL
LIN {X 0,Y 321.04,Z 774.562,A -85,B 0,C 180,E1 -11825.84,E2 -11825.84} C_VEL
LIN {X 0,Y 322.437,Z 765.346,A -85,B 0,C 180,E1 -11826.564,E2 -11826.564} C_VEL
LIN {X 0,Y 322.704,Z 759.329,A -85,B 0,C 180,E1 -11827.077,E2 -11827.077} C_VEL
LIN {X 0,Y 320.008,Z 741.916,A -85,B 0,C 180,E1 -11828.807,E2 -11828.807} C_VEL
LIN {X 0,Y 319.594,Z 734.654,A -85,B 0,C 180,E1 -11829.284,E2 -11829.284} C_VEL
LIN {X 0,Y 319.638,Z 733.578,A -85,B 0,C 180,E1 -11829.33,E2 -11829.33} C_VEL
LIN {X 0,Y 320.517,Z 713.99,A -85,B 0,C 180,E1 -11829.992,E2 -11829.992} C_VEL
LIN {X 0,Y 323.405,Z 645.82,A -85,B 0,C 180,E1 -11831.535,E2 -11831.535} C_VEL
LIN {X 0,Y 329.508,Z 519.039,A -85,B 0,C 180,E1 -11834.303,E2 -11834.303} C_VEL
LIN {X 0,Y 328.961,Z 514.428,A -85,B 0,C 180,E1 -11834.54,E2 -11834.54} C_VEL
LIN {X 0,Y 325.997,Z 516.415,A -85,B 0,C 180,E1 -11835.011,E2 -11835.011} C_VEL
LIN {X 0,Y 324.199,Z 516.503,A -85,B 0,C 180,E1 -11835.351,E2 -11835.351} C_VEL
LIN {X 0,Y 316.744,Z 559.974,A -85,B 0,C 180,E1 -11840.147,E2 -11840.147} C_VEL
LIN {X 0,Y 309.795,Z 605.576,A -85,B 0,C 180,E1 -11845.161,E2 -11845.161} C_VEL
LIN {X 0,Y 308.384,Z 616.59,A -85,B 0,C 180,E1 -11846.321,E2 -11846.321} C_VEL
LIN {X 0,Y 308.638,Z 626.594,A -85,B 0,C 180,E1 -11846.804,E2 -11846.804} C_VEL
LIN {X 0,Y 299.948,Z 729.652,A -85,B 0,C 180,E1 -11850.685,E2 -11850.685} C_VEL
LIN {X 0,Y 297.366,Z 769.673,A -85,B 0,C 180,E1 -11852.435,E2 -11852.435} C_VEL
LIN {X 0,Y 295.956,Z 788.122,A -85,B 0,C 180,E1 -11853.623,E2 -11853.623} C_VEL
LIN {X 0,Y 294.254,Z 804.644,A -85,B 0,C 180,E1 -11855.08,E2 -11855.08} C_VEL
LIN {X 0,Y 292.351,Z 820.213,A -85,B 0,C 180,E1 -11856.839,E2 -11856.839} C_VEL
LIN {X 0,Y 290.285,Z 835.446,A -85,B 0,C 180,E1 -11859.009,E2 -11859.009} C_VEL
LIN {X 0,Y 288.327,Z 848.855,A -85,B 0,C 180,E1 -11861.395,E2 -11861.395} C_VEL
LIN {X 0,Y 286.599,Z 860.779,A -85,B 0,C 180,E1 -11864.001,E2 -11864.001} C_VEL
LIN {X 0,Y 285.079,Z 871.842,A -85,B 0,C 180,E1 -11867.028,E2 -11867.028} C_VEL
LIN {X 0,Y 284.027,Z 880.6,A -85,B 0,C 180,E1 -11870.067,E2 -11870.067} C_VEL
LIN {X 0,Y 283.399,Z 887.91,A -85,B 0,C 180,E1 -11873.313,E2 -11873.313} C_VEL
LIN {X 0,Y 283.224,Z 893.548,A -85,B 0,C 180,E1 -11876.761,E2 -11876.761} C_VEL
LIN {X 0,Y 283.494,Z 897.104,A -85,B 0,C 180,E1 -11879.999,E2 -11879.999} C_VEL
LIN {X 0,Y 284.221,Z 899.127,A -85,B 0,C 180,E1 -11883.428,E2 -11883.428} C_VEL
LIN {X 0,Y 285.496,Z 899.345,A -85,B 0,C 180,E1 -11886.838,E2 -11886.838} C_VEL
LIN {X 0,Y 287.422,Z 897.869,A -85,B 0,C 180,E1 -11890.219,E2 -11890.219} C_VEL
LIN {X 0,Y 290.257,Z 894.387,A -85,B 0,C 180,E1 -11893.749,E2 -11893.749} C_VEL
LIN {X 0,Y 293.935,Z 888.872,A -85,B 0,C 180,E1 -11897.213,E2 -11897.213} C_VEL
LIN {X 0,Y 298.554,Z 881.193,A -85,B 0,C 180,E1 -11900.587,E2 -11900.587} C_VEL
LIN {X 0,Y 303.806,Z 871.746,A -85,B 0,C 180,E1 -11903.672,E2 -11903.672} C_VEL
LIN {X 0,Y 309.582,Z 860.696,A -85,B 0,C 180,E1 -11906.467,E2 -11906.467} C_VEL
LIN {X 0,Y 315.849,Z 848.36,A -85,B 0,C 180,E1 -11908.969,E2 -11908.969} C_VEL
LIN {X 0,Y 323.612,Z 832.847,A -85,B 0,C 180,E1 -11911.476,E2 -11911.476} C_VEL
LIN {X 0,Y 332.202,Z 816.026,A -85,B 0,C 180,E1 -11913.628,E2 -11913.628} C_VEL
LIN {X 0,Y 343.011,Z 796.76,A -85,B 0,C 180,E1 -11915.582,E2 -11915.582} C_VEL
LIN {X 0,Y 352.331,Z 780.848,A -85,B 0,C 180,E1 -11916.911,E2 -11916.911} C_VEL
LIN {X 0,Y 342.042,Z 803.294,A -85,B 0,C 180,E1 -11918.559,E2 -11918.559} C_VEL
LIN {X 0,Y 331.618,Z 826.023,A -85,B 0,C 180,E1 -11920.685,E2 -11920.685} C_VEL
LIN {X 0,Y 321.025,Z 849.915,A -85,B 0,C 180,E1 -11923.472,E2 -11923.472} C_VEL
LIN {X 0,Y 311.474,Z 872.375,A -85,B 0,C 180,E1 -11926.686,E2 -11926.686} C_VEL
LIN {X 0,Y 302.939,Z 893.962,A -85,B 0,C 180,E1 -11930.431,E2 -11930.431} C_VEL
LIN {X 0,Y 295.819,Z 913.645,A -85,B 0,C 180,E1 -11934.544,E2 -11934.544} C_VEL
LIN {X 0,Y 290.242,Z 930.876,A -85,B 0,C 180,E1 -11938.886,E2 -11938.886} C_VEL
LIN {X 0,Y 286.092,Z 945.753,A -85,B 0,C 180,E1 -11943.426,E2 -11943.426} C_VEL
LIN {X 0,Y 283.421,Z 957.541,A -85,B 0,C 180,E1 -11947.822,E2 -11947.822} C_VEL
LIN {X 0,Y 281.89,Z 966.682,A -85,B 0,C 180,E1 -11952.025,E2 -11952.025} C_VEL
LIN {X 0,Y 281.178,Z 973.926,A -85,B 0,C 180,E1 -11956.216,E2 -11956.216} C_VEL
LIN {X 0,Y 281.048,Z 979.261,A -85,B 0,C 180,E1 -11960.374,E2 -11960.374} C_VEL
LIN {X 0,Y 281.225,Z 982.519,A -85,B 0,C 180,E1 -11964.081,E2 -11964.081} C_VEL
LIN {X 0,Y 281.384,Z 984.237,A -85,B 0,C 180,E1 -11967.759,E2 -11967.759} C_VEL
LIN {X 0,Y 281.418,Z 984.489,A -85,B 0,C 180,E1 -11971.221,E2 -11971.221} C_VEL
LIN {X 0,Y 281.269,Z 983.38,A -85,B 0,C 180,E1 -11974.689,E2 -11974.689} C_VEL
LIN {X 0,Y 281.093,Z 980.684,A -85,B 0,C 180,E1 -11978.385,E2 -11978.385} C_VEL
LIN {X 0,Y 281.102,Z 976.174,A -85,B 0,C 180,E1 -11982.322,E2 -11982.322} C_VEL
LIN {X 0,Y 281.578,Z 969.845,A -85,B 0,C 180,E1 -11986.291,E2 -11986.291} C_VEL
LIN {X 0,Y 282.691,Z 961.648,A -85,B 0,C 180,E1 -11990.28,E2 -11990.28} C_VEL
LIN {X 0,Y 284.618,Z 951.425,A -85,B 0,C 180,E1 -11994.268,E2 -11994.268} C_VEL
LIN {X 0,Y 287.473,Z 938.951,A -85,B 0,C 180,E1 -11998.23,E2 -11998.23} C_VEL
LIN {X 0,Y 291.107,Z 924.754,A -85,B 0,C 180,E1 -12001.933,E2 -12001.933} C_VEL
LIN {X 0,Y 295.391,Z 908.887,A -85,B 0,C 180,E1 -12005.366,E2 -12005.366} C_VEL
LIN {X 0,Y 300.225,Z 891.348,A -85,B 0,C 180,E1 -12008.519,E2 -12008.519} C_VEL
LIN {X 0,Y 305.109,Z 873.447,A -85,B 0,C 180,E1 -12011.199,E2 -12011.199} C_VEL
LIN {X 0,Y 310.207,Z 854.11,A -85,B 0,C 180,E1 -12013.611,E2 -12013.611} C_VEL
LIN {X 0,Y 315.152,Z 834.212,A -85,B 0,C 180,E1 -12015.666,E2 -12015.666} C_VEL
LIN {X 0,Y 320.252,Z 812.211,A -85,B 0,C 180,E1 -12017.529,E2 -12017.529} C_VEL
LIN {X 0,Y 324.689,Z 790.995,A -85,B 0,C 180,E1 -12018.978,E2 -12018.978} C_VEL
LIN {X 0,Y 328.903,Z 767.788,A -85,B 0,C 180,E1 -12020.206,E2 -12020.206} C_VEL
LIN {X 0,Y 332.145,Z 744.913,A -85,B 0,C 180,E1 -12021.118,E2 -12021.118} C_VEL
LIN {X 0,Y 334.87,Z 719.135,A -85,B 0,C 180,E1 -12021.866,E2 -12021.866} C_VEL
LIN {X 0,Y 337.723,Z 700.314,A -85,B 0,C 180,E1 -12022.23,E2 -12022.23} C_VEL
LIN {X 0,Y 350.4,Z 671.555,A -85,B 0,C 180,E1 -12023.717,E2 -12023.717} C_VEL
LIN {X 0,Y 361.153,Z 649.879,A -85,B 0,C 180,E1 -12024.619,E2 -12024.619} C_VEL
LIN {X 0,Y 365.467,Z 641.736,A -85,B 0,C 180,E1 -12024.911,E2 -12024.911} C_VEL
LIN {X 0,Y 360.238,Z 623.651,A -85,B 0,C 180,E1 -12027.61,E2 -12027.61} C_VEL
LIN {X 0,Y 357.081,Z 603.581,A -85,B 0,C 180,E1 -12030.382,E2 -12030.382} C_VEL
LIN {X 0,Y 356.204,Z 582.64,A -85,B 0,C 180,E1 -12033.043,E2 -12033.043} C_VEL
LIN {X 0,Y 357.58,Z 559.38,A -85,B 0,C 180,E1 -12035.73,E2 -12035.73} C_VEL
LIN {X 0,Y 361.13,Z 534.854,A -85,B 0,C 180,E1 -12038.266,E2 -12038.266} C_VEL
LIN {X 0,Y 352.541,Z 517.952,A -85,B 0,C 180,E1 -12042.334,E2 -12042.334} C_VEL
LIN {X 0,Y 345.046,Z 503.945,A -85,B 0,C 180,E1 -12046.084,E2 -12046.084} C_VEL
LIN {X 0,Y 338.178,Z 491.216,A -85,B 0,C 180,E1 -12049.782,E2 -12049.782} C_VEL
LIN {X 0,Y 330.7,Z 477.756,A -85,B 0,C 180,E1 -12054.105,E2 -12054.105} C_VEL
LIN {X 0,Y 324.535,Z 467.047,A -85,B 0,C 180,E1 -12057.882,E2 -12057.882} C_VEL
LIN {X 0,Y 319.066,Z 457.495,A -85,B 0,C 180,E1 -12061.528,E2 -12061.528} C_VEL
LIN {X 0,Y 314.01,Z 448.699,A -85,B 0,C 180,E1 -12065.116,E2 -12065.116} C_VEL
LIN {X 0,Y 310.012,Z 442.149,A -85,B 0,C 180,E1 -12068.053,E2 -12068.053} C_VEL
LIN {X 0,Y 307.598,Z 437.947,A -85,B 0,C 180,E1 -12069.968,E2 -12069.968} C_VEL
LIN {X 0,Y 304.477,Z 432.689,A -85,B 0,C 180,E1 -12072.518,E2 -12072.518} C_VEL
LIN {X 0,Y 301.431,Z 427.521,A -85,B 0,C 180,E1 -12075.149,E2 -12075.149} C_VEL
LIN {X 0,Y 298.589,Z 422.647,A -85,B 0,C 180,E1 -12077.742,E2 -12077.742} C_VEL
LIN {X 0,Y 296.027,Z 418.389,A -85,B 0,C 180,E1 -12080.153,E2 -12080.153} C_VEL
LIN {X 0,Y 293.073,Z 413.307,A -85,B 0,C 180,E1 -12083.313,E2 -12083.313} C_VEL
LIN {X 0,Y 294.718,Z 413.294,A -85,B 0,C 180,E1 -12084.024,E2 -12084.024} C_VEL
LIN {X 0,Y 297.946,Z 418.376,A -85,B 0,C 180,E1 -12086.08,E2 -12086.08} C_VEL
LIN {X 0,Y 299.18,Z 420.334,A -85,B 0,C 180,E1 -12086.819,E2 -12086.819} C_VEL
LIN {X 0,Y 302.345,Z 425.404,A -85,B 0,C 180,E1 -12088.654,E2 -12088.654} C_VEL
LIN {X 0,Y 305.573,Z 430.988,A -85,B 0,C 180,E1 -12090.476,E2 -12090.476} C_VEL
LIN {X 0,Y 309.982,Z 438.645,A -85,B 0,C 180,E1 -12092.813,E2 -12092.813} C_VEL
LIN {X 0,Y 315.901,Z 450.346,A -85,B 0,C 180,E1 -12095.879,E2 -12095.879} C_VEL
LIN {X 0,Y 321.889,Z 463.496,A -85,B 0,C 180,E1 -12098.863,E2 -12098.863} C_VEL
LIN {X 0,Y 327.687,Z 478.514,A -85,B 0,C 180,E1 -12101.814,E2 -12101.814} C_VEL
LIN {X 0,Y 330.861,Z 487.514,A -85,B 0,C 180,E1 -12103.399,E2 -12103.399} C_VEL
LIN {X 0,Y 328.926,Z 514.065,A -85,B 0,C 180,E1 -12105.565,E2 -12105.565} C_VEL
LIN {X 0,Y 329.451,Z 521.614,A -85,B 0,C 180,E1 -12105.887,E2 -12105.887} C_VEL
LIN {X 0,Y 320.499,Z 711.544,A -85,B 0,C 180,E1 -12110.053,E2 -12110.053} C_VEL
LIN {X 0,Y 319.66,Z 731.813,A -85,B 0,C 180,E1 -12110.707,E2 -12110.707} C_VEL
LIN {X 0,Y 318.114,Z 750.211,A -85,B 0,C 180,E1 -12111.608,E2 -12111.608} C_VEL
LIN {X 0,Y 315.842,Z 768.025,A -85,B 0,C 180,E1 -12112.797,E2 -12112.797} C_VEL
LIN {X 0,Y 312.844,Z 785.583,A -85,B 0,C 180,E1 -12114.319,E2 -12114.319} C_VEL
LIN {X 0,Y 309.401,Z 802.105,A -85,B 0,C 180,E1 -12116.153,E2 -12116.153} C_VEL
LIN {X 0,Y 305.691,Z 817.125,A -85,B 0,C 180,E1 -12118.224,E2 -12118.224} C_VEL
LIN {X 0,Y 301.733,Z 831.276,A -85,B 0,C 180,E1 -12120.636,E2 -12120.636} C_VEL
LIN {X 0,Y 297.893,Z 843.84,A -85,B 0,C 180,E1 -12123.272,E2 -12123.272} C_VEL
LIN {X 0,Y 294.261,Z 854.975,A -85,B 0,C 180,E1 -12126.15,E2 -12126.15} C_VEL
LIN {X 0,Y 290.975,Z 864.701,A -85,B 0,C 180,E1 -12129.273,E2 -12129.273} C_VEL
LIN {X 0,Y 288.015,Z 873.426,A -85,B 0,C 180,E1 -12132.838,E2 -12132.838} C_VEL
LIN {X 0,Y 285.769,Z 880.152,A -85,B 0,C 180,E1 -12136.443,E2 -12136.443} C_VEL
LIN {X 0,Y 284.217,Z 885.094,A -85,B 0,C 180,E1 -12140.074,E2 -12140.074} C_VEL
LIN {X 0,Y 283.237,Z 888.553,A -85,B 0,C 180,E1 -12143.921,E2 -12143.921} C_VEL
LIN {X 0,Y 282.764,Z 890.332,A -85,B 0,C 180,E1 -12147.771,E2 -12147.771} C_VEL
LIN {X 0,Y 282.723,Z 890.489,A -85,B 0,C 180,E1 -12151.622,E2 -12151.622} C_VEL
LIN {X 0,Y 283.123,Z 889.03,A -85,B 0,C 180,E1 -12155.472,E2 -12155.472} C_VEL
LIN {X 0,Y 284.007,Z 885.911,A -85,B 0,C 180,E1 -12159.32,E2 -12159.32} C_VEL
LIN {X 0,Y 285.531,Z 880.987,A -85,B 0,C 180,E1 -12163.157,E2 -12163.157} C_VEL
LIN {X 0,Y 287.683,Z 874.517,A -85,B 0,C 180,E1 -12166.767,E2 -12166.767} C_VEL
LIN {X 0,Y 290.369,Z 866.611,A -85,B 0,C 180,E1 -12170.142,E2 -12170.142} C_VEL
LIN {X 0,Y 293.525,Z 857.317,A -85,B 0,C 180,E1 -12173.275,E2 -12173.275} C_VEL
LIN {X 0,Y 297.045,Z 846.672,A -85,B 0,C 180,E1 -12176.165,E2 -12176.165} C_VEL
LIN {X 0,Y 300.782,Z 834.667,A -85,B 0,C 180,E1 -12178.817,E2 -12178.817} C_VEL
LIN {X 0,Y 304.643,Z 821.218,A -85,B 0,C 180,E1 -12181.237,E2 -12181.237} C_VEL
LIN {X 0,Y 308.321,Z 806.919,A -85,B 0,C 180,E1 -12183.335,E2 -12183.335} C_VEL
LIN {X 0,Y 311.697,Z 791.68,A -85,B 0,C 180,E1 -12185.156,E2 -12185.156} C_VEL
LIN {X 0,Y 314.665,Z 775.792,A -85,B 0,C 180,E1 -12186.683,E2 -12186.683} C_VEL
LIN {X 0,Y 317.131,Z 759.254,A -85,B 0,C 180,E1 -12187.938,E2 -12187.938} C_VEL
LIN {X 0,Y 319.053,Z 741.182,A -85,B 0,C 180,E1 -12188.98,E2 -12188.98} C_VEL
LIN {X 0,Y 319.638,Z 733.578,A -85,B 0,C 180,E1 -12189.33,E2 -12189.33} C_VEL
LIN {X 0,Y 319.377,Z 726.133,A -85,B 0,C 180,E1 -12189.732,E2 -12189.732} C_VEL
LIN {X 0,Y 315.467,Z 707.676,A -85,B 0,C 180,E1 -12190.991,E2 -12190.991} C_VEL
LIN {X 0,Y 314.944,Z 700.137,A -85,B 0,C 180,E1 -12191.296,E2 -12191.296} C_VEL
LIN {X 0,Y 323.428,Z 529.147,A -85,B 0,C 180,E1 -12195.083,E2 -12195.083} C_VEL
LIN {X 0,Y 318.89,Z 534.518,A -85,B 0,C 180,E1 -12195.762,E2 -12195.762} C_VEL
LIN {X 0,Y 316.346,Z 536.269,A -85,B 0,C 180,E1 -12196.196,E2 -12196.196} C_VEL
LIN {X 0,Y 314.532,Z 536.539,A -85,B 0,C 180,E1 -12196.572,E2 -12196.572} C_VEL
LIN {X 0,Y 306.988,Z 580.964,A -85,B 0,C 180,E1 -12201.531,E2 -12201.531} C_VEL
LIN {X 0,Y 301.561,Z 617.36,A -85,B 0,C 180,E1 -12205.541,E2 -12205.541} C_VEL
LIN {X 0,Y 301.786,Z 627.36,A -85,B 0,C 180,E1 -12206.035,E2 -12206.035} C_VEL
LIN {X 0,Y 292.377,Z 734.153,A -85,B 0,C 180,E1 -12210.195,E2 -12210.195} C_VEL
LIN {X 0,Y 289.878,Z 771.616,A -85,B 0,C 180,E1 -12211.926,E2 -12211.926} C_VEL
LIN {X 0,Y 288.449,Z 789.137,A -85,B 0,C 180,E1 -12213.104,E2 -12213.104} C_VEL
LIN {X 0,Y 286.573,Z 806.589,A -85,B 0,C 180,E1 -12214.696,E2 -12214.696} C_VEL
LIN {X 0,Y 284.65,Z 821.688,A -85,B 0,C 180,E1 -12216.462,E2 -12216.462} C_VEL
LIN {X 0,Y 282.483,Z 837.122,A -85,B 0,C 180,E1 -12218.727,E2 -12218.727} C_VEL
LIN {X 0,Y 280.395,Z 850.951,A -85,B 0,C 180,E1 -12221.28,E2 -12221.28} C_VEL
LIN {X 0,Y 278.633,Z 862.674,A -85,B 0,C 180,E1 -12223.959,E2 -12223.959} C_VEL
LIN {X 0,Y 277.098,Z 873.648,A -85,B 0,C 180,E1 -12227.072,E2 -12227.072} C_VEL
LIN {X 0,Y 276.001,Z 882.858,A -85,B 0,C 180,E1 -12230.407,E2 -12230.407} C_VEL
LIN {X 0,Y 275.446,Z 889.581,A -85,B 0,C 180,E1 -12233.538,E2 -12233.538} C_VEL
LIN {X 0,Y 275.318,Z 895.208,A -85,B 0,C 180,E1 -12237.097,E2 -12237.097} C_VEL
LIN {X 0,Y 275.689,Z 898.887,A -85,B 0,C 180,E1 -12240.623,E2 -12240.623} C_VEL
LIN {X 0,Y 276.577,Z 900.819,A -85,B 0,C 180,E1 -12244.146,E2 -12244.146} C_VEL
LIN {X 0,Y 278.155,Z 900.919,A -85,B 0,C 180,E1 -12247.85,E2 -12247.85} C_VEL
LIN {X 0,Y 280.377,Z 899.245,A -85,B 0,C 180,E1 -12251.311,E2 -12251.311} C_VEL
LIN {X 0,Y 283.381,Z 895.889,A -85,B 0,C 180,E1 -12254.716,E2 -12254.716} C_VEL
LIN {X 0,Y 287.585,Z 890.186,A -85,B 0,C 180,E1 -12258.348,E2 -12258.348} C_VEL
LIN {X 0,Y 292.494,Z 882.779,A -85,B 0,C 180,E1 -12261.665,E2 -12261.665} C_VEL
LIN {X 0,Y 298.204,Z 873.51,A -85,B 0,C 180,E1 -12264.778,E2 -12264.778} C_VEL
LIN {X 0,Y 304.474,Z 862.798,A -85,B 0,C 180,E1 -12267.582,E2 -12267.582} C_VEL
LIN {X 0,Y 311.748,Z 850.141,A -85,B 0,C 180,E1 -12270.234,E2 -12270.234} C_VEL
LIN {X 0,Y 320.778,Z 834.349,A -85,B 0,C 180,E1 -12272.843,E2 -12272.843} C_VEL
LIN {X 0,Y 330.487,Z 817.785,A -85,B 0,C 180,E1 -12274.981,E2 -12274.981} C_VEL
LIN {X 0,Y 342.169,Z 799.517,A -85,B 0,C 180,E1 -12276.869,E2 -12276.869} C_VEL
LIN {X 0,Y 330.778,Z 821.94,A -85,B 0,C 180,E1 -12278.889,E2 -12278.889} C_VEL
LIN {X 0,Y 319.225,Z 845.181,A -85,B 0,C 180,E1 -12281.531,E2 -12281.531} C_VEL
LIN {X 0,Y 308.339,Z 867.902,A -85,B 0,C 180,E1 -12284.752,E2 -12284.752} C_VEL
LIN {X 0,Y 298.727,Z 889.461,A -85,B 0,C 180,E1 -12288.492,E2 -12288.492} C_VEL
LIN {X 0,Y 290.844,Z 908.743,A -85,B 0,C 180,E1 -12292.519,E2 -12292.519} C_VEL
LIN {X 0,Y 284.851,Z 924.97,A -85,B 0,C 180,E1 -12296.558,E2 -12296.558} C_VEL
LIN {X 0,Y 280.244,Z 939.117,A -85,B 0,C 180,E1 -12300.738,E2 -12300.738} C_VEL
LIN {X 0,Y 276.651,Z 952.289,A -85,B 0,C 180,E1 -12305.44,E2 -12305.44} C_VEL
LIN {X 0,Y 274.484,Z 962.671,A -85,B 0,C 180,E1 -12310.018,E2 -12310.018} C_VEL
LIN {X 0,Y 273.432,Z 970.411,A -85,B 0,C 180,E1 -12314.3,E2 -12314.3} C_VEL
LIN {X 0,Y 273.097,Z 976.408,A -85,B 0,C 180,E1 -12318.597,E2 -12318.597} C_VEL
LIN {X 0,Y 273.202,Z 980.355,A -85,B 0,C 180,E1 -12322.653,E2 -12322.653} C_VEL
LIN {X 0,Y 273.432,Z 982.569,A -85,B 0,C 180,E1 -12326.435,E2 -12326.435} C_VEL
LIN {X 0,Y 273.537,Z 983.284,A -85,B 0,C 180,E1 -12329.999,E2 -12329.999} C_VEL
LIN {X 0,Y 273.445,Z 982.569,A -85,B 0,C 180,E1 -12333.563,E2 -12333.563} C_VEL
LIN {X 0,Y 273.227,Z 980.312,A -85,B 0,C 180,E1 -12337.358,E2 -12337.358} C_VEL
LIN {X 0,Y 273.147,Z 976.504,A -85,B 0,C 180,E1 -12341.186,E2 -12341.186} C_VEL
LIN {X 0,Y 273.481,Z 970.366,A -85,B 0,C 180,E1 -12345.479,E2 -12345.479} C_VEL
LIN {X 0,Y 274.461,Z 962.588,A -85,B 0,C 180,E1 -12349.581,E2 -12349.581} C_VEL
LIN {X 0,Y 276.142,Z 953.38,A -85,B 0,C 180,E1 -12353.471,E2 -12353.471} C_VEL
LIN {X 0,Y 278.661,Z 942.209,A -85,B 0,C 180,E1 -12357.34,E2 -12357.34} C_VEL
LIN {X 0,Y 282.1,Z 928.826,A -85,B 0,C 180,E1 -12361.162,E2 -12361.162} C_VEL
LIN {X 0,Y 286.23,Z 913.832,A -85,B 0,C 180,E1 -12364.707,E2 -12364.707} C_VEL
LIN {X 0,Y 291.043,Z 896.854,A -85,B 0,C 180,E1 -12368.036,E2 -12368.036} C_VEL
LIN {X 0,Y 296.258,Z 878.445,A -85,B 0,C 180,E1 -12371.027,E2 -12371.027} C_VEL
LIN {X 0,Y 301.934,Z 857.677,A -85,B 0,C 180,E1 -12373.796,E2 -12373.796} C_VEL
LIN {X 0,Y 307.346,Z 837.02,A -85,B 0,C 180,E1 -12376.067,E2 -12376.067} C_VEL
LIN {X 0,Y 312.414,Z 816.177,A -85,B 0,C 180,E1 -12377.944,E2 -12377.944} C_VEL
LIN {X 0,Y 317.279,Z 793.942,A -85,B 0,C 180,E1 -12379.543,E2 -12379.543} C_VEL
LIN {X 0,Y 321.606,Z 771.491,A -85,B 0,C 180,E1 -12380.807,E2 -12380.807} C_VEL
LIN {X 0,Y 325.374,Z 747.148,A -85,B 0,C 180,E1 -12381.851,E2 -12381.851} C_VEL
LIN {X 0,Y 328.269,Z 721.085,A -85,B 0,C 180,E1 -12382.661,E2 -12382.661} C_VEL
LIN {X 0,Y 331.638,Z 699.253,A -85,B 0,C 180,E1 -12383.101,E2 -12383.101} C_VEL
LIN {X 0,Y 344.651,Z 670.2,A -85,B 0,C 180,E1 -12384.607,E2 -12384.607} C_VEL
LIN {X 0,Y 355.921,Z 647.946,A -85,B 0,C 180,E1 -12385.538,E2 -12385.538} C_VEL
LIN {X 0,Y 358.327,Z 643.552,A -85,B 0,C 180,E1 -12385.692,E2 -12385.692} C_VEL
LIN {X 0,Y 353.318,Z 624.56,A -85,B 0,C 180,E1 -12388.526,E2 -12388.526} C_VEL
LIN {X 0,Y 350.567,Z 603.997,A -85,B 0,C 180,E1 -12391.37,E2 -12391.37} C_VEL
LIN {X 0,Y 350.108,Z 582.406,A -85,B 0,C 180,E1 -12394.104,E2 -12394.104} C_VEL
LIN {X 0,Y 351.94,Z 558.698,A -85,B 0,C 180,E1 -12396.829,E2 -12396.829} C_VEL
LIN {X 0,Y 355.038,Z 539.134,A -85,B 0,C 180,E1 -12398.871,E2 -12398.871} C_VEL
LIN {X 0,Y 346.684,Z 522.635,A -85,B 0,C 180,E1 -12402.892,E2 -12402.892} C_VEL
LIN {X 0,Y 338.33,Z 506.782,A -85,B 0,C 180,E1 -12407.195,E2 -12407.195} C_VEL
LIN {X 0,Y 330.588,Z 492.65,A -85,B 0,C 180,E1 -12411.478,E2 -12411.478} C_VEL
LIN {X 0,Y 323.209,Z 479.312,A -85,B 0,C 180,E1 -12415.92,E2 -12415.92} C_VEL
LIN {X 0,Y 316.278,Z 467.319,A -85,B 0,C 180,E1 -12420.363,E2 -12420.363} C_VEL
LIN {X 0,Y 311.523,Z 459.052,A -85,B 0,C 180,E1 -12423.681,E2 -12423.681} C_VEL
LIN {X 0,Y 308.108,Z 453.333,A -85,B 0,C 180,E1 -12426.148,E2 -12426.148} C_VEL
LIN {X 0,Y 305.338,Z 448.521,A -85,B 0,C 180,E1 -12428.285,E2 -12428.285} C_VEL
LIN {X 0,Y 302.82,Z 444.17,A -85,B 0,C 180,E1 -12430.283,E2 -12430.283} C_VEL
LIN {X 0,Y 299.883,Z 439.158,A -85,B 0,C 180,E1 -12432.713,E2 -12432.713} C_VEL
LIN {X 0,Y 296.751,Z 433.863,A -85,B 0,C 180,E1 -12435.438,E2 -12435.438} C_VEL
LIN {X 0,Y 293.944,Z 429.035,A -85,B 0,C 180,E1 -12438.032,E2 -12438.032} C_VEL
LIN {X 0,Y 291.404,Z 424.68,A -85,B 0,C 180,E1 -12440.495,E2 -12440.495} C_VEL
LIN {X 0,Y 289.073,Z 421.172,A -85,B 0,C 180,E1 -12442.793,E2 -12442.793} C_VEL
LIN {X 0,Y 291.747,Z 421.047,A -85,B 0,C 180,E1 -12443.962,E2 -12443.962} C_VEL
LIN {X 0,Y 294.48,Z 425.397,A -85,B 0,C 180,E1 -12445.761,E2 -12445.761} C_VEL
LIN {X 0,Y 298.493,Z 432.099,A -85,B 0,C 180,E1 -12448.242,E2 -12448.242} C_VEL
LIN {X 0,Y 303.507,Z 440.905,A -85,B 0,C 180,E1 -12451.146,E2 -12451.146} C_VEL
LIN {X 0,Y 309.191,Z 451.824,A -85,B 0,C 180,E1 -12454.242,E2 -12454.242} C_VEL
LIN {X 0,Y 315.702,Z 466.074,A -85,B 0,C 180,E1 -12457.68,E2 -12457.68} C_VEL
LIN {X 0,Y 321.612,Z 481.086,A -85,B 0,C 180,E1 -12460.759,E2 -12460.759} C_VEL
LIN {X 0,Y 325.1,Z 491.62,A -85,B 0,C 180,E1 -12462.646,E2 -12462.646} C_VEL
LIN {X 0,Y 323.294,Z 515.321,A -85,B 0,C 180,E1 -12464.581,E2 -12464.581} C_VEL
LIN {X 0,Y 323.789,Z 522.762,A -85,B 0,C 180,E1 -12464.907,E2 -12464.907} C_VEL
LIN {X 0,Y 314.474,Z 712.049,A -85,B 0,C 180,E1 -12469.107,E2 -12469.107} C_VEL
LIN {X 0,Y 313.587,Z 732.715,A -85,B 0,C 180,E1 -12469.778,E2 -12469.778} C_VEL
LIN {X 0,Y 311.985,Z 751.131,A -85,B 0,C 180,E1 -12470.688,E2 -12470.688} C_VEL
LIN {X 0,Y 309.763,Z 768.041,A -85,B 0,C 180,E1 -12471.821,E2 -12471.821} C_VEL
LIN {X 0,Y 306.752,Z 785.255,A -85,B 0,C 180,E1 -12473.307,E2 -12473.307} C_VEL
LIN {X 0,Y 303.262,Z 801.648,A -85,B 0,C 180,E1 -12475.109,E2 -12475.109} C_VEL
LIN {X 0,Y 299.335,Z 817.2,A -85,B 0,C 180,E1 -12477.24,E2 -12477.24} C_VEL
LIN {X 0,Y 295.179,Z 831.553,A -85,B 0,C 180,E1 -12479.689,E2 -12479.689} C_VEL
LIN {X 0,Y 291.086,Z 844.404,A -85,B 0,C 180,E1 -12482.402,E2 -12482.402} C_VEL
LIN {X 0,Y 287.276,Z 855.577,A -85,B 0,C 180,E1 -12485.314,E2 -12485.314} C_VEL
LIN {X 0,Y 283.777,Z 865.427,A -85,B 0,C 180,E1 -12488.505,E2 -12488.505} C_VEL
LIN {X 0,Y 280.744,Z 873.883,A -85,B 0,C 180,E1 -12491.975,E2 -12491.975} C_VEL
LIN {X 0,Y 278.298,Z 880.762,A -85,B 0,C 180,E1 -12495.647,E2 -12495.647} C_VEL
LIN {X 0,Y 276.478,Z 886.181,A -85,B 0,C 180,E1 -12499.633,E2 -12499.633} C_VEL
LIN {X 0,Y 275.412,Z 889.671,A -85,B 0,C 180,E1 -12503.539,E2 -12503.539} C_VEL
LIN {X 0,Y 274.881,Z 891.532,A -85,B 0,C 180,E1 -12507.499,E2 -12507.499} C_VEL
LIN {X 0,Y 274.815,Z 891.773,A -85,B 0,C 180,E1 -12511.46,E2 -12511.46} C_VEL
LIN {X 0,Y 275.229,Z 890.36,A -85,B 0,C 180,E1 -12515.496,E2 -12515.496} C_VEL
LIN {X 0,Y 276.129,Z 887.366,A -85,B 0,C 180,E1 -12519.378,E2 -12519.378} C_VEL
LIN {X 0,Y 277.718,Z 882.565,A -85,B 0,C 180,E1 -12523.322,E2 -12523.322} C_VEL
LIN {X 0,Y 279.961,Z 876.209,A -85,B 0,C 180,E1 -12527.03,E2 -12527.03} C_VEL
LIN {X 0,Y 282.94,Z 867.874,A -85,B 0,C 180,E1 -12530.695,E2 -12530.695} C_VEL
LIN {X 0,Y 286.264,Z 858.578,A -85,B 0,C 180,E1 -12533.902,E2 -12533.902} C_VEL
LIN {X 0,Y 289.959,Z 847.93,A -85,B 0,C 180,E1 -12536.855,E2 -12536.855} C_VEL
LIN {X 0,Y 293.874,Z 835.921,A -85,B 0,C 180,E1 -12539.561,E2 -12539.561} C_VEL
LIN {X 0,Y 297.909,Z 822.468,A -85,B 0,C 180,E1 -12542.026,E2 -12542.026} C_VEL
LIN {X 0,Y 301.765,Z 808.096,A -85,B 0,C 180,E1 -12544.168,E2 -12544.168} C_VEL
LIN {X 0,Y 305.231,Z 793.105,A -85,B 0,C 180,E1 -12545.99,E2 -12545.99} C_VEL
LIN {X 0,Y 308.362,Z 777.021,A -85,B 0,C 180,E1 -12547.56,E2 -12547.56} C_VEL
LIN {X 0,Y 311.048,Z 759.532,A -85,B 0,C 180,E1 -12548.896,E2 -12548.896} C_VEL
LIN {X 0,Y 313.027,Z 741.298,A -85,B 0,C 180,E1 -12549.944,E2 -12549.944} C_VEL
LIN {X 0,Y 314.229,Z 722.025,A -85,B 0,C 180,E1 -12550.716,E2 -12550.716} C_VEL
LIN {X 0,Y 314.944,Z 700.137,A -85,B 0,C 180,E1 -12551.296,E2 -12551.296} C_VEL
LIN {X 0,Y 314.517,Z 692.556,A -85,B 0,C 180,E1 -12551.598,E2 -12551.598} C_VEL
LIN {X 0,Y 310.927,Z 672.731,A -85,B 0,C 180,E1 -12552.828,E2 -12552.828} C_VEL
LIN {X 0,Y 310.726,Z 666.212,A -85,B 0,C 180,E1 -12553.069,E2 -12553.069} C_VEL
LIN {X 0,Y 317.128,Z 543.917,A -85,B 0,C 180,E1 -12555.795,E2 -12555.795} C_VEL
LIN {X 0,Y 310.967,Z 552.964,A -85,B 0,C 180,E1 -12556.711,E2 -12556.711} C_VEL
LIN {X 0,Y 307.3,Z 556.522,A -85,B 0,C 180,E1 -12557.344,E2 -12557.344} C_VEL
LIN {X 0,Y 305.051,Z 557.218,A -85,B 0,C 180,E1 -12557.797,E2 -12557.797} C_VEL
LIN {X 0,Y 304.705,Z 557.195,A -85,B 0,C 180,E1 -12557.883,E2 -12557.883} C_VEL
LIN {X 0,Y 297.14,Z 602.184,A -85,B 0,C 180,E1 -12562.963,E2 -12562.963} C_VEL
LIN {X 0,Y 294.793,Z 618.349,A -85,B 0,C 180,E1 -12564.74,E2 -12564.74} C_VEL
LIN {X 0,Y 294.947,Z 628.138,A -85,B 0,C 180,E1 -12565.242,E2 -12565.242} C_VEL
LIN {X 0,Y 285.82,Z 727.017,A -85,B 0,C 180,E1 -12569.192,E2 -12569.192} C_VEL
LIN {X 0,Y 282.646,Z 769.854,A -85,B 0,C 180,E1 -12571.192,E2 -12571.192} C_VEL
LIN {X 0,Y 281.214,Z 787.467,A -85,B 0,C 180,E1 -12572.354,E2 -12572.354} C_VEL
LIN {X 0,Y 279.374,Z 804.633,A -85,B 0,C 180,E1 -12573.882,E2 -12573.882} C_VEL
LIN {X 0,Y 277.201,Z 821.423,A -85,B 0,C 180,E1 -12575.833,E2 -12575.833} C_VEL
LIN {X 0,Y 274.961,Z 836.769,A -85,B 0,C 180,E1 -12578.115,E2 -12578.115} C_VEL
LIN {X 0,Y 272.928,Z 849.886,A -85,B 0,C 180,E1 -12580.526,E2 -12580.526} C_VEL
LIN {X 0,Y 270.914,Z 862.919,A -85,B 0,C 180,E1 -12583.489,E2 -12583.489} C_VEL
LIN {X 0,Y 269.29,Z 874.099,A -85,B 0,C 180,E1 -12586.69,E2 -12586.69} C_VEL
LIN {X 0,Y 268.183,Z 883.003,A -85,B 0,C 180,E1 -12589.907,E2 -12589.907} C_VEL
LIN {X 0,Y 267.537,Z 890.449,A -85,B 0,C 180,E1 -12593.346,E2 -12593.346} C_VEL
LIN {X 0,Y 267.398,Z 896.256,A -85,B 0,C 180,E1 -12596.999,E2 -12596.999} C_VEL
LIN {X 0,Y 267.761,Z 900.009,A -85,B 0,C 180,E1 -12600.427,E2 -12600.427} C_VEL
LIN {X 0,Y 268.737,Z 902.312,A -85,B 0,C 180,E1 -12604.267,E2 -12604.267} C_VEL
LIN {X 0,Y 270.301,Z 902.676,A -85,B 0,C 180,E1 -12607.866,E2 -12607.866} C_VEL
LIN {X 0,Y 272.632,Z 901.404,A -85,B 0,C 180,E1 -12611.422,E2 -12611.422} C_VEL
LIN {X 0,Y 275.975,Z 898.187,A -85,B 0,C 180,E1 -12615.12,E2 -12615.12} C_VEL
LIN {X 0,Y 280.277,Z 893.041,A -85,B 0,C 180,E1 -12618.727,E2 -12618.727} C_VEL
LIN {X 0,Y 285.282,Z 886.341,A -85,B 0,C 180,E1 -12622.025,E2 -12622.025} C_VEL
LIN {X 0,Y 291.254,Z 877.78,A -85,B 0,C 180,E1 -12625.193,E2 -12625.193} C_VEL
LIN {X 0,Y 298.256,Z 867.27,A -85,B 0,C 180,E1 -12628.208,E2 -12628.208} C_VEL
LIN {X 0,Y 306.368,Z 854.652,A -85,B 0,C 180,E1 -12631.04,E2 -12631.04} C_VEL
LIN {X 0,Y 315.874,Z 840.04,A -85,B 0,C 180,E1 -12633.637,E2 -12633.637} C_VEL
LIN {X 0,Y 326.341,Z 824.372,A -85,B 0,C 180,E1 -12635.816,E2 -12635.816} C_VEL
LIN {X 0,Y 332.374,Z 815.704,A -85,B 0,C 180,E1 -12636.827,E2 -12636.827} C_VEL
LIN {X 0,Y 319.68,Z 838.527,A -85,B 0,C 180,E1 -12639.275,E2 -12639.275} C_VEL
LIN {X 0,Y 308.121,Z 859.757,A -85,B 0,C 180,E1 -12642.141,E2 -12642.141} C_VEL
LIN {X 0,Y 297.137,Z 881.147,A -85,B 0,C 180,E1 -12645.701,E2 -12645.701} C_VEL
LIN {X 0,Y 287.324,Z 901.966,A -85,B 0,C 180,E1 -12649.925,E2 -12649.925} C_VEL
LIN {X 0,Y 279.377,Z 920.793,A -85,B 0,C 180,E1 -12654.564,E2 -12654.564} C_VEL
LIN {X 0,Y 273.607,Z 936.43,A -85,B 0,C 180,E1 -12659.228,E2 -12659.228} C_VEL
LIN {X 0,Y 269.491,Z 949.692,A -85,B 0,C 180,E1 -12664.036,E2 -12664.036} C_VEL
LIN {X 0,Y 266.958,Z 960.149,A -85,B 0,C 180,E1 -12668.696,E2 -12668.696} C_VEL
LIN {X 0,Y 265.646,Z 968.214,A -85,B 0,C 180,E1 -12673.152,E2 -12673.152} C_VEL
LIN {X 0,Y 265.148,Z 974.683,A -85,B 0,C 180,E1 -12677.808,E2 -12677.808} C_VEL
LIN {X 0,Y 265.234,Z 978.767,A -85,B 0,C 180,E1 -12681.982,E2 -12681.982} C_VEL
LIN {X 0,Y 265.492,Z 981.12,A -85,B 0,C 180,E1 -12685.896,E2 -12685.896} C_VEL
LIN {X 0,Y 265.629,Z 981.953,A -85,B 0,C 180,E1 -12689.568,E2 -12689.568} C_VEL
LIN {X 0,Y 265.569,Z 981.353,A -85,B 0,C 180,E1 -12693.237,E2 -12693.237} C_VEL
LIN {X 0,Y 265.345,Z 979.334,A -85,B 0,C 180,E1 -12696.925,E2 -12696.925} C_VEL
LIN {X 0,Y 265.23,Z 975.684,A -85,B 0,C 180,E1 -12700.864,E2 -12700.864} C_VEL
LIN {X 0,Y 265.478,Z 970.021,A -85,B 0,C 180,E1 -12705.062,E2 -12705.062} C_VEL
LIN {X 0,Y 266.327,Z 962.95,A -85,B 0,C 180,E1 -12709.063,E2 -12709.063} C_VEL
LIN {X 0,Y 268.114,Z 953.109,A -85,B 0,C 180,E1 -12713.454,E2 -12713.454} C_VEL
LIN {X 0,Y 270.869,Z 941.2,A -85,B 0,C 180,E1 -12717.716,E2 -12717.716} C_VEL
LIN {X 0,Y 274.429,Z 927.782,A -85,B 0,C 180,E1 -12721.644,E2 -12721.644} C_VEL
LIN {X 0,Y 278.843,Z 912.277,A -85,B 0,C 180,E1 -12725.386,E2 -12725.386} C_VEL
LIN {X 0,Y 283.744,Z 895.579,A -85,B 0,C 180,E1 -12728.717,E2 -12728.717} C_VEL
LIN {X 0,Y 289.081,Z 877.259,A -85,B 0,C 180,E1 -12731.744,E2 -12731.744} C_VEL
LIN {X 0,Y 294.952,Z 856.419,A -85,B 0,C 180,E1 -12734.564,E2 -12734.564} C_VEL
LIN {X 0,Y 300.351,Z 836.376,A -85,B 0,C 180,E1 -12736.806,E2 -12736.806} C_VEL
LIN {X 0,Y 305.749,Z 814.851,A -85,B 0,C 180,E1 -12738.776,E2 -12738.776} C_VEL
LIN {X 0,Y 310.824,Z 792.289,A -85,B 0,C 180,E1 -12740.416,E2 -12740.416} C_VEL
LIN {X 0,Y 315.307,Z 769.527,A -85,B 0,C 180,E1 -12741.705,E2 -12741.705} C_VEL
LIN {X 0,Y 319.053,Z 745.772,A -85,B 0,C 180,E1 -12742.732,E2 -12742.732} C_VEL
LIN {X 0,Y 322.094,Z 719.632,A -85,B 0,C 180,E1 -12743.55,E2 -12743.55} C_VEL
LIN {X 0,Y 325.639,Z 698.101,A -85,B 0,C 180,E1 -12744.004,E2 -12744.004} C_VEL
LIN {X 0,Y 339.416,Z 667.968,A -85,B 0,C 180,E1 -12745.571,E2 -12745.571} C_VEL
LIN {X 0,Y 351.116,Z 645.214,A -85,B 0,C 180,E1 -12746.495,E2 -12746.495} C_VEL
LIN {X 0,Y 346.32,Z 624.687,A -85,B 0,C 180,E1 -12749.557,E2 -12749.557} C_VEL
LIN {X 0,Y 344.031,Z 603.516,A -85,B 0,C 180,E1 -12752.478,E2 -12752.478} C_VEL
LIN {X 0,Y 344.115,Z 581.445,A -85,B 0,C 180,E1 -12755.267,E2 -12755.267} C_VEL
LIN {X 0,Y 346.45,Z 557.917,A -85,B 0,C 180,E1 -12757.965,E2 -12757.965} C_VEL
LIN {X 0,Y 348.793,Z 543.145,A -85,B 0,C 180,E1 -12759.53,E2 -12759.53} C_VEL
LIN {X 0,Y 340.819,Z 527.272,A -85,B 0,C 180,E1 -12763.467,E2 -12763.467} C_VEL
LIN {X 0,Y 332.451,Z 511.429,A -85,B 0,C 180,E1 -12767.847,E2 -12767.847} C_VEL
LIN {X 0,Y 325.283,Z 498.252,A -85,B 0,C 180,E1 -12771.872,E2 -12771.872} C_VEL
LIN {X 0,Y 318.165,Z 485.305,A -85,B 0,C 180,E1 -12776.217,E2 -12776.217} C_VEL
LIN {X 0,Y 311.528,Z 473.705,A -85,B 0,C 180,E1 -12780.552,E2 -12780.552} C_VEL
LIN {X 0,Y 306.418,Z 464.855,A -85,B 0,C 180,E1 -12784.117,E2 -12784.117} C_VEL
LIN {X 0,Y 303.255,Z 459.505,A -85,B 0,C 180,E1 -12786.437,E2 -12786.437} C_VEL
LIN {X 0,Y 300.472,Z 454.647,A -85,B 0,C 180,E1 -12788.613,E2 -12788.613} C_VEL
LIN {X 0,Y 297.727,Z 449.92,A -85,B 0,C 180,E1 -12790.84,E2 -12790.84} C_VEL
LIN {X 0,Y 295.034,Z 445.263,A -85,B 0,C 180,E1 -12793.125,E2 -12793.125} C_VEL
LIN {X 0,Y 292.136,Z 440.279,A -85,B 0,C 180,E1 -12795.688,E2 -12795.688} C_VEL
LIN {X 0,Y 289.29,Z 435.404,A -85,B 0,C 180,E1 -12798.332,E2 -12798.332} C_VEL
LIN {X 0,Y 285.97,Z 429.902,A -85,B 0,C 180,E1 -12801.539,E2 -12801.539} C_VEL
LIN {X 0,Y 285.263,Z 428.854,A -85,B 0,C 180,E1 -12802.314,E2 -12802.314} C_VEL
LIN {X 0,Y 288.536,Z 428.692,A -85,B 0,C 180,E1 -12803.819,E2 -12803.819} C_VEL
LIN {X 0,Y 291.765,Z 433.963,A -85,B 0,C 180,E1 -12806.018,E2 -12806.018} C_VEL
LIN {X 0,Y 294.771,Z 439.059,A -85,B 0,C 180,E1 -12807.911,E2 -12807.911} C_VEL
LIN {X 0,Y 299.48,Z 447.469,A -85,B 0,C 180,E1 -12810.719,E2 -12810.719} C_VEL
LIN {X 0,Y 304.658,Z 457.713,A -85,B 0,C 180,E1 -12813.687,E2 -12813.687} C_VEL
LIN {X 0,Y 310.759,Z 471.425,A -85,B 0,C 180,E1 -12817.068,E2 -12817.068} C_VEL
LIN {X 0,Y 316.641,Z 486.612,A -85,B 0,C 180,E1 -12820.223,E2 -12820.223} C_VEL
LIN {X 0,Y 319.451,Z 495.22,A -85,B 0,C 180,E1 -12821.812,E2 -12821.812} C_VEL
LIN {X 0,Y 317.756,Z 516.541,A -85,B 0,C 180,E1 -12823.561,E2 -12823.561} C_VEL
LIN {X 0,Y 318.218,Z 524.035,A -85,B 0,C 180,E1 -12823.896,E2 -12823.896} C_VEL
LIN {X 0,Y 308.537,Z 712.546,A -85,B 0,C 180,E1 -12828.125,E2 -12828.125} C_VEL
LIN {X 0,Y 307.601,Z 733.621,A -85,B 0,C 180,E1 -12828.813,E2 -12828.813} C_VEL
LIN {X 0,Y 305.928,Z 752.156,A -85,B 0,C 180,E1 -12829.737,E2 -12829.737} C_VEL
LIN {X 0,Y 303.588,Z 769.282,A -85,B 0,C 180,E1 -12830.899,E2 -12830.899} C_VEL
LIN {X 0,Y 300.454,Z 786.496,A -85,B 0,C 180,E1 -12832.406,E2 -12832.406} C_VEL
LIN {X 0,Y 296.991,Z 802.126,A -85,B 0,C 180,E1 -12834.141,E2 -12834.141} C_VEL
LIN {X 0,Y 293.063,Z 817.184,A -85,B 0,C 180,E1 -12836.213,E2 -12836.213} C_VEL
LIN {X 0,Y 288.896,Z 831.154,A -85,B 0,C 180,E1 -12838.582,E2 -12838.582} C_VEL
LIN {X 0,Y 284.711,Z 843.891,A -85,B 0,C 180,E1 -12841.242,E2 -12841.242} C_VEL
LIN {X 0,Y 280.612,Z 855.488,A -85,B 0,C 180,E1 -12844.234,E2 -12844.234} C_VEL
LIN {X 0,Y 276.849,Z 865.609,A -85,B 0,C 180,E1 -12847.492,E2 -12847.492} C_VEL
LIN {X 0,Y 273.577,Z 874.244,A -85,B 0,C 180,E1 -12851.018,E2 -12851.018} C_VEL
LIN {X 0,Y 270.884,Z 881.372,A -85,B 0,C 180,E1 -12854.808,E2 -12854.808} C_VEL
LIN {X 0,Y 268.964,Z 886.688,A -85,B 0,C 180,E1 -12858.638,E2 -12858.638} C_VEL
LIN {X 0,Y 267.691,Z 890.498,A -85,B 0,C 180,E1 -12862.705,E2 -12862.705} C_VEL
LIN {X 0,Y 267.04,Z 892.61,A -85,B 0,C 180,E1 -12866.781,E2 -12866.781} C_VEL
LIN {X 0,Y 266.9,Z 893.096,A -85,B 0,C 180,E1 -12870.859,E2 -12870.859} C_VEL
LIN {X 0,Y 267.24,Z 891.973,A -85,B 0,C 180,E1 -12874.937,E2 -12874.937} C_VEL
LIN {X 0,Y 268.119,Z 889.201,A -85,B 0,C 180,E1 -12879.012,E2 -12879.012} C_VEL
